LIN {X 0,Y 190.941,Z 458.891,A -85,B 0,C 180,E1 -21861.534,E2 -21861.534} C_VEL
LIN {X 0,Y 190.385,Z 460.614,A -85,B 0,C 180,E1 -21865.766,E2 -21865.766} C_VEL
LIN {X 0,Y 190.301,Z 461.211,A -85,B 0,C 180,E1 -21870,E2 -21870} C_VEL
LIN {X 0,Y 190.444,Z 460.499,A -85,B 0,C 180,E1 -21874.869,E2 -21874.869} C_VEL
LIN {X 0,Y 190.929,Z 458.975,A -85,B 0,C 180,E1 -21878.467,E2 -21878.467} C_VEL
LIN {X 0,Y 192.019,Z 456.147,A -85,B 0,C 180,E1 -21882.686,E2 -21882.686} C_VEL
LIN {X 0,Y 193.845,Z 452.093,A -85,B 0,C 180,E1 -21886.861,E2 -21886.861} C_VEL
LIN {X 0,Y 196.509,Z 446.712,A -85,B 0,C 180,E1 -21890.956,E2 -21890.956} C_VEL
LIN {X 0,Y 199.993,Z 439.849,A -85,B 0,C 180,E1 -21894.942,E2 -21894.942} C_VEL
LIN {X 0,Y 204.393,Z 431.274,A -85,B 0,C 180,E1 -21898.776,E2 -21898.776} C_VEL
LIN {X 0,Y 208.235,Z 423.562,A -85,B 0,C 180,E1 -21901.543,E2 -21901.543} C_VEL
LIN {X 0,Y 213.047,Z 412.865,A -85,B 0,C 180,E1 -21904.684,E2 -21904.684} C_VEL
LIN {X 0,Y 217.826,Z 401.819,A -85,B 0,C 180,E1 -21907.226,E2 -21907.226} C_VEL
LIN {X 0,Y 222.415,Z 389.72,A -85,B 0,C 180,E1 -21909.489,E2 -21909.489} C_VEL
LIN {X 0,Y 226.964,Z 376.424,A -85,B 0,C 180,E1 -21911.444,E2 -21911.444} C_VEL
LIN {X 0,Y 230.741,Z 362.87,A -85,B 0,C 180,E1 -21913.049,E2 -21913.049} C_VEL
LIN {X 0,Y 233.967,Z 349.116,A -85,B 0,C 180,E1 -21914.299,E2 -21914.299} C_VEL
LIN {X 0,Y 236.667,Z 334.427,A -85,B 0,C 180,E1 -21915.304,E2 -21915.304} C_VEL
LIN {X 0,Y 238.709,Z 319.352,A -85,B 0,C 180,E1 -21916.012,E2 -21916.012} C_VEL
LIN {X 0,Y 240.388,Z 297.392,A -85,B 0,C 180,E1 -21916.657,E2 -21916.657} C_VEL
LIN {X 0,Y 244.269,Z 236.804,A -85,B 0,C 180,E1 -21918.261,E2 -21918.261} C_VEL
LIN {X 0,Y 244.011,Z 235.536,A -85,B 0,C 180,E1 -21918.384,E2 -21918.384} C_VEL
LIN {X 0,Y 240.281,Z 227.752,A -85,B 0,C 180,E1 -21919.755,E2 -21919.755} C_VEL
LIN {X 0,Y 233.168,Z 215.506,A -85,B 0,C 180,E1 -21922.485,E2 -21922.485} C_VEL
LIN {X 0,Y 226.96,Z 205.762,A -85,B 0,C 180,E1 -21925.117,E2 -21925.117} C_VEL
LIN {X 0,Y 220.972,Z 197.115,A -85,B 0,C 180,E1 -21927.944,E2 -21927.944} C_VEL
LIN {X 0,Y 217.819,Z 192.871,A -85,B 0,C 180,E1 -21929.574,E2 -21929.574} C_VEL
LIN {X 0,Y 214.771,Z 188.838,A -85,B 0,C 180,E1 -21931.274,E2 -21931.274} C_VEL
LIN {X 0,Y 211.806,Z 184.879,A -85,B 0,C 180,E1 -21933.076,E2 -21933.076} C_VEL
LIN {X 0,Y 208.608,Z 181.315,A -85,B 0,C 180,E1 -21935.161,E2 -21935.161} C_VEL
LIN {X 0,Y 207.472,Z 179.38,A -85,B 0,C 180,E1 -21936.015,E2 -21936.015} C_VEL
LIN {X 0,Y 204.831,Z 177.101,A -85,B 0,C 180,E1 -21937.958,E2 -21937.958} C_VEL
LIN {X 0,Y 202.842,Z 173.863,A -85,B 0,C 180,E1 -21939.728,E2 -21939.728} C_VEL
LIN {X 0,Y 200.216,Z 171.989,A -85,B 0,C 180,E1 -21942.109,E2 -21942.109} C_VEL
LIN {X 0,Y 198.473,Z 169.066,A -85,B 0,C 180,E1 -21944.138,E2 -21944.138} C_VEL
LIN {X 0,Y 198.172,Z 168.139,A -85,B 0,C 180,E1 -21944.575,E2 -21944.575} C_VEL
LIN {X 0,Y 195.147,Z 166.479,A -85,B 0,C 180,E1 -21948.575,E2 -21948.575} C_VEL
LIN {X 0,Y 193.085,Z 162.801,A -85,B 0,C 180,E1 -21953.337,E2 -21953.337} C_VEL
LIN {X 0,Y 192.962,Z 162.066,A -85,B 0,C 180,E1 -21953.989,E2 -21953.989} C_VEL
LIN {X 0,Y 193.233,Z 162.041,A -85,B 0,C 180,E1 -21957.915,E2 -21957.915} C_VEL
LIN {X 0,Y 193.418,Z 162.001,A -85,B 0,C 180,E1 -21960,E2 -21960} C_VEL
LIN {X 0,Y 192.961,Z 162.06,A -85,B 0,C 180,E1 -21964.177,E2 -21964.177} C_VEL
LIN {X 0,Y 192.994,Z 162.232,A -85,B 0,C 180,E1 -21965.878,E2 -21965.878} C_VEL
LIN {X 0,Y 193.886,Z 164.688,A -85,B 0,C 180,E1 -21968.599,E2 -21968.599} C_VEL
LIN {X 0,Y 196.209,Z 167.297,A -85,B 0,C 180,E1 -21972.673,E2 -21972.673} C_VEL
LIN {X 0,Y 198.286,Z 168.3,A -85,B 0,C 180,E1 -21975.219,E2 -21975.219} C_VEL
LIN {X 0,Y 199.512,Z 170.977,A -85,B 0,C 180,E1 -21976.776,E2 -21976.776} C_VEL
LIN {X 0,Y 201.821,Z 173.285,A -85,B 0,C 180,E1 -21979.054,E2 -21979.054} C_VEL
LIN {X 0,Y 203.195,Z 174.283,A -85,B 0,C 180,E1 -21980.235,E2 -21980.235} C_VEL
LIN {X 0,Y 205.071,Z 177.346,A -85,B 0,C 180,E1 -21981.882,E2 -21981.882} C_VEL
LIN {X 0,Y 207.81,Z 179.895,A -85,B 0,C 180,E1 -21983.889,E2 -21983.889} C_VEL
LIN {X 0,Y 210.275,Z 183.372,A -85,B 0,C 180,E1 -21985.62,E2 -21985.62} C_VEL
LIN {X 0,Y 211.91,Z 185.069,A -85,B 0,C 180,E1 -21986.645,E2 -21986.645} C_VEL
LIN {X 0,Y 214.922,Z 189.001,A -85,B 0,C 180,E1 -21988.462,E2 -21988.462} C_VEL
LIN {X 0,Y 219.469,Z 195.238,A -85,B 0,C 180,E1 -21990.955,E2 -21990.955} C_VEL
LIN {X 0,Y 223.648,Z 202.088,A -85,B 0,C 180,E1 -21993.079,E2 -21993.079} C_VEL
LIN {X 0,Y 225.037,Z 204.616,A -85,B 0,C 180,E1 -21993.757,E2 -21993.757} C_VEL
LIN {X 0,Y 226.117,Z 207.654,A -85,B 0,C 180,E1 -21994.329,E2 -21994.329} C_VEL
LIN {X 0,Y 227.686,Z 214.53,A -85,B 0,C 180,E1 -21995.267,E2 -21995.267} C_VEL
LIN {X 0,Y 229.607,Z 223.383,A -85,B 0,C 180,E1 -21996.393,E2 -21996.393} C_VEL
LIN {X 0,Y 231.422,Z 228.024,A -85,B 0,C 180,E1 -21997.227,E2 -21997.227} C_VEL
LIN {X 0,Y 236.293,Z 238.89,A -85,B 0,C 180,E1 -21999.258,E2 -21999.258} C_VEL
LIN {X 0,Y 239.067,Z 245.621,A -85,B 0,C 180,E1 -22000.365,E2 -22000.365} C_VEL
LIN {X 0,Y 233.645,Z 325.426,A -85,B 0,C 180,E1 -22002.527,E2 -22002.527} C_VEL
LIN {X 0,Y 231.489,Z 341.56,A -85,B 0,C 180,E1 -22003.227,E2 -22003.227} C_VEL
LIN {X 0,Y 228.504,Z 356.805,A -85,B 0,C 180,E1 -22004.191,E2 -22004.191} C_VEL
LIN {X 0,Y 224.971,Z 370.535,A -85,B 0,C 180,E1 -22005.34,E2 -22005.34} C_VEL
LIN {X 0,Y 220.972,Z 384.002,A -85,B 0,C 180,E1 -22006.859,E2 -22006.859} C_VEL
LIN {X 0,Y 216.181,Z 397.756,A -85,B 0,C 180,E1 -22008.84,E2 -22008.84} C_VEL
LIN {X 0,Y 211.132,Z 410.12,A -85,B 0,C 180,E1 -22011.075,E2 -22011.075} C_VEL
LIN {X 0,Y 205.65,Z 422.297,A -85,B 0,C 180,E1 -22013.877,E2 -22013.877} C_VEL
LIN {X 0,Y 201.168,Z 431.703,A -85,B 0,C 180,E1 -22016.617,E2 -22016.617} C_VEL
LIN {X 0,Y 196.664,Z 440.962,A -85,B 0,C 180,E1 -22019.98,E2 -22019.98} C_VEL
LIN {X 0,Y 192.028,Z 449.677,A -85,B 0,C 180,E1 -22023.948,E2 -22023.948} C_VEL
LIN {X 0,Y 188.492,Z 456.683,A -85,B 0,C 180,E1 -22028.108,E2 -22028.108} C_VEL
LIN {X 0,Y 185.856,Z 462.197,A -85,B 0,C 180,E1 -22032.391,E2 -22032.391} C_VEL
LIN {X 0,Y 184.088,Z 466.373,A -85,B 0,C 180,E1 -22036.758,E2 -22036.758} C_VEL
LIN {X 0,Y 183.224,Z 469.308,A -85,B 0,C 180,E1 -22041.174,E2 -22041.174} C_VEL
LIN {X 0,Y 182.976,Z 471.063,A -85,B 0,C 180,E1 -22045.594,E2 -22045.594} C_VEL
LIN {X 0,Y 183.168,Z 471.669,A -85,B 0,C 180,E1 -22050,E2 -22050} C_VEL
LIN {X 0,Y 182.976,Z 471.047,A -85,B 0,C 180,E1 -22054.406,E2 -22054.406} C_VEL
LIN {X 0,Y 183.224,Z 469.271,A -85,B 0,C 180,E1 -22058.826,E2 -22058.826} C_VEL
LIN {X 0,Y 184.079,Z 466.319,A -85,B 0,C 180,E1 -22063.243,E2 -22063.243} C_VEL
LIN {X 0,Y 185.81,Z 462.128,A -85,B 0,C 180,E1 -22067.613,E2 -22067.613} C_VEL
LIN {X 0,Y 188.416,Z 456.587,A -85,B 0,C 180,E1 -22071.901,E2 -22071.901} C_VEL
LIN {X 0,Y 191.989,Z 449.551,A -85,B 0,C 180,E1 -22076.058,E2 -22076.058} C_VEL
LIN {X 0,Y 196.011,Z 442.038,A -85,B 0,C 180,E1 -22079.538,E2 -22079.538} C_VEL
LIN {X 0,Y 200.409,Z 432.978,A -85,B 0,C 180,E1 -22082.925,E2 -22082.925} C_VEL
LIN {X 0,Y 205.637,Z 422.094,A -85,B 0,C 180,E1 -22086.125,E2 -22086.125} C_VEL
LIN {X 0,Y 211.082,Z 409.864,A -85,B 0,C 180,E1 -22088.936,E2 -22088.936} C_VEL
LIN {X 0,Y 216.189,Z 397.432,A -85,B 0,C 180,E1 -22091.163,E2 -22091.163} C_VEL
LIN {X 0,Y 220.929,Z 383.607,A -85,B 0,C 180,E1 -22093.151,E2 -22093.151} C_VEL
LIN {X 0,Y 224.965,Z 370.042,A -85,B 0,C 180,E1 -22094.661,E2 -22094.661} C_VEL
LIN {X 0,Y 228.465,Z 356.243,A -85,B 0,C 180,E1 -22095.819,E2 -22095.819} C_VEL
LIN {X 0,Y 231.35,Z 341.579,A -85,B 0,C 180,E1 -22096.73,E2 -22096.73} C_VEL
LIN {X 0,Y 233.473,Z 325.428,A -85,B 0,C 180,E1 -22097.439,E2 -22097.439} C_VEL
LIN {X 0,Y 237.987,Z 259.996,A -85,B 0,C 180,E1 -22099.205,E2 -22099.205} C_VEL
LIN {X 0,Y 238.911,Z 245.472,A -85,B 0,C 180,E1 -22099.603,E2 -22099.603} C_VEL
LIN {X 0,Y 233.217,Z 231.952,A -85,B 0,C 180,E1 -22101.916,E2 -22101.916} C_VEL
LIN {X 0,Y 227.378,Z 220.017,A -85,B 0,C 180,E1 -22104.446,E2 -22104.446} C_VEL
LIN {X 0,Y 221.444,Z 208.914,A -85,B 0,C 180,E1 -22107.279,E2 -22107.279} C_VEL
LIN {X 0,Y 215.755,Z 199.426,A -85,B 0,C 180,E1 -22110.304,E2 -22110.304} C_VEL
LIN {X 0,Y 212.344,Z 194.903,A -85,B 0,C 180,E1 -22112.262,E2 -22112.262} C_VEL
LIN {X 0,Y 209.046,Z 190.532,A -85,B 0,C 180,E1 -22114.352,E2 -22114.352} C_VEL
LIN {X 0,Y 206.249,Z 187.049,A -85,B 0,C 180,E1 -22116.294,E2 -22116.294} C_VEL
LIN {X 0,Y 205.535,Z 185.913,A -85,B 0,C 180,E1 -22116.845,E2 -22116.845} C_VEL
LIN {X 0,Y 202.873,Z 183.255,A -85,B 0,C 180,E1 -22118.903,E2 -22118.903} C_VEL
LIN {X 0,Y 201.286,Z 180.606,A -85,B 0,C 180,E1 -22120.363,E2 -22120.363} C_VEL
LIN {X 0,Y 198.766,Z 178.632,A -85,B 0,C 180,E1 -22122.715,E2 -22122.715} C_VEL
LIN {X 0,Y 196.966,Z 175.504,A -85,B 0,C 180,E1 -22124.876,E2 -22124.876} C_VEL
LIN {X 0,Y 196.681,Z 175.002,A -85,B 0,C 180,E1 -22125.251,E2 -22125.251} C_VEL
LIN {X 0,Y 193.832,Z 173.17,A -85,B 0,C 180,E1 -22129.159,E2 -22129.159} C_VEL
LIN {X 0,Y 192.097,Z 169.801,A -85,B 0,C 180,E1 -22133.171,E2 -22133.171} C_VEL
LIN {X 0,Y 191.96,Z 169.223,A -85,B 0,C 180,E1 -22133.694,E2 -22133.694} C_VEL
LIN {X 0,Y 190.794,Z 168.603,A -85,B 0,C 180,E1 -22140,E2 -22140} C_VEL
LIN {X 0,Y 191.988,Z 169.275,A -85,B 0,C 180,E1 -22146.833,E2 -22146.833} C_VEL
LIN {X 0,Y 193.266,Z 172.44,A -85,B 0,C 180,E1 -22150.233,E2 -22150.233} C_VEL
LIN {X 0,Y 195.81,Z 174.67,A -85,B 0,C 180,E1 -22154.153,E2 -22154.153} C_VEL
LIN {X 0,Y 196.855,Z 175.279,A -85,B 0,C 180,E1 -22155.415,E2 -22155.415} C_VEL
LIN {X 0,Y 198.677,Z 178.613,A -85,B 0,C 180,E1 -22157.641,E2 -22157.641} C_VEL
LIN {X 0,Y 201.497,Z 180.984,A -85,B 0,C 180,E1 -22160.28,E2 -22160.28} C_VEL
LIN {X 0,Y 203.639,Z 184.293,A -85,B 0,C 180,E1 -22162.178,E2 -22162.178} C_VEL
LIN {X 0,Y 205.866,Z 186.424,A -85,B 0,C 180,E1 -22163.849,E2 -22163.849} C_VEL
LIN {X 0,Y 208.48,Z 190.012,A -85,B 0,C 180,E1 -22165.724,E2 -22165.724} C_VEL
LIN {X 0,Y 209.841,Z 191.608,A -85,B 0,C 180,E1 -22166.613,E2 -22166.613} C_VEL
LIN {X 0,Y 213.845,Z 196.934,A -85,B 0,C 180,E1 -22169.064,E2 -22169.064} C_VEL
LIN {X 0,Y 218.027,Z 202.706,A -85,B 0,C 180,E1 -22171.362,E2 -22171.362} C_VEL
LIN {X 0,Y 223.276,Z 210.46,A -85,B 0,C 180,E1 -22173.967,E2 -22173.967} C_VEL
LIN {X 0,Y 228.709,Z 219.049,A -85,B 0,C 180,E1 -22176.403,E2 -22176.403} C_VEL
LIN {X 0,Y 235.134,Z 230.2,A -85,B 0,C 180,E1 -22179.027,E2 -22179.027} C_VEL
LIN {X 0,Y 238.764,Z 237.398,A -85,B 0,C 180,E1 -22180.428,E2 -22180.428} C_VEL
LIN {X 0,Y 239.308,Z 238.724,A -85,B 0,C 180,E1 -22180.642,E2 -22180.642} C_VEL
LIN {X 0,Y 233.946,Z 317.1,A -85,B 0,C 180,E1 -22182.766,E2 -22182.766} C_VEL
LIN {X 0,Y 231.838,Z 333.001,A -85,B 0,C 180,E1 -22183.477,E2 -22183.477} C_VEL
LIN {X 0,Y 229.059,Z 348.105,A -85,B 0,C 180,E1 -22184.491,E2 -22184.491} C_VEL
LIN {X 0,Y 226.025,Z 361.087,A -85,B 0,C 180,E1 -22185.657,E2 -22185.657} C_VEL
LIN {X 0,Y 221.867,Z 375.842,A -85,B 0,C 180,E1 -22187.383,E2 -22187.383} C_VEL
LIN {X 0,Y 217.118,Z 389.289,A -85,B 0,C 180,E1 -22189.35,E2 -22189.35} C_VEL
LIN {X 0,Y 212.28,Z 401.491,A -85,B 0,C 180,E1 -22191.628,E2 -22191.628} C_VEL
LIN {X 0,Y 207.292,Z 412.609,A -85,B 0,C 180,E1 -22194.208,E2 -22194.208} C_VEL
LIN {X 0,Y 202.289,Z 423.39,A -85,B 0,C 180,E1 -22197.418,E2 -22197.418} C_VEL
LIN {X 0,Y 197.636,Z 432.347,A -85,B 0,C 180,E1 -22200.728,E2 -22200.728} C_VEL
LIN {X 0,Y 193.637,Z 439.764,A -85,B 0,C 180,E1 -22204.181,E2 -22204.181} C_VEL
LIN {X 0,Y 189.901,Z 446.69,A -85,B 0,C 180,E1 -22208.279,E2 -22208.279} C_VEL
LIN {X 0,Y 187.08,Z 452.124,A -85,B 0,C 180,E1 -22212.51,E2 -22212.51} C_VEL
LIN {X 0,Y 185.133,Z 456.219,A -85,B 0,C 180,E1 -22216.834,E2 -22216.834} C_VEL
LIN {X 0,Y 183.898,Z 459.091,A -85,B 0,C 180,E1 -22221.207,E2 -22221.207} C_VEL
LIN {X 0,Y 183.308,Z 460.812,A -85,B 0,C 180,E1 -22225.602,E2 -22225.602} C_VEL
LIN {X 0,Y 183.207,Z 461.41,A -85,B 0,C 180,E1 -22230,E2 -22230} C_VEL
LIN {X 0,Y 183.331,Z 460.795,A -85,B 0,C 180,E1 -22234.645,E2 -22234.645} C_VEL
LIN {X 0,Y 183.882,Z 459.174,A -85,B 0,C 180,E1 -22238.794,E2 -22238.794} C_VEL
LIN {X 0,Y 185.084,Z 456.345,A -85,B 0,C 180,E1 -22243.17,E2 -22243.17} C_VEL
LIN {X 0,Y 187.046,Z 452.292,A -85,B 0,C 180,E1 -22247.493,E2 -22247.493} C_VEL
LIN {X 0,Y 189.867,Z 446.91,A -85,B 0,C 180,E1 -22251.725,E2 -22251.725} C_VEL
LIN {X 0,Y 193.541,Z 440.048,A -85,B 0,C 180,E1 -22255.833,E2 -22255.833} C_VEL
LIN {X 0,Y 198.166,Z 431.472,A -85,B 0,C 180,E1 -22259.77,E2 -22259.77} C_VEL
LIN {X 0,Y 202.904,Z 422.349,A -85,B 0,C 180,E1 -22263.061,E2 -22263.061} C_VEL
LIN {X 0,Y 207.227,Z 413.062,A -85,B 0,C 180,E1 -22265.805,E2 -22265.805} C_VEL
LIN {X 0,Y 212.212,Z 402.015,A -85,B 0,C 180,E1 -22268.386,E2 -22268.386} C_VEL
LIN {X 0,Y 216.97,Z 389.915,A -85,B 0,C 180,E1 -22270.684,E2 -22270.684} C_VEL
LIN {X 0,Y 221.696,Z 376.618,A -85,B 0,C 180,E1 -22272.658,E2 -22272.658} C_VEL
LIN {X 0,Y 225.536,Z 363.341,A -85,B 0,C 180,E1 -22274.247,E2 -22274.247} C_VEL
LIN {X 0,Y 228.938,Z 349.308,A -85,B 0,C 180,E1 -22275.54,E2 -22275.54} C_VEL
LIN {X 0,Y 231.744,Z 334.615,A -85,B 0,C 180,E1 -22276.548,E2 -22276.548} C_VEL
LIN {X 0,Y 233.836,Z 319.536,A -85,B 0,C 180,E1 -22277.263,E2 -22277.263} C_VEL
LIN {X 0,Y 235.572,Z 297.567,A -85,B 0,C 180,E1 -22277.912,E2 -22277.912} C_VEL
LIN {X 0,Y 239.422,Z 238.711,A -85,B 0,C 180,E1 -22279.499,E2 -22279.499} C_VEL
LIN {X 0,Y 236.266,Z 232.138,A -85,B 0,C 180,E1 -22280.719,E2 -22280.719} C_VEL
LIN {X 0,Y 229.894,Z 220.899,A -85,B 0,C 180,E1 -22283.289,E2 -22283.289} C_VEL
LIN {X 0,Y 223.643,Z 210.885,A -85,B 0,C 180,E1 -22286.072,E2 -22286.072} C_VEL
LIN {X 0,Y 218.192,Z 202.869,A -85,B 0,C 180,E1 -22288.776,E2 -22288.776} C_VEL
LIN {X 0,Y 214.91,Z 198.382,A -85,B 0,C 180,E1 -22290.56,E2 -22290.56} C_VEL
LIN {X 0,Y 212.446,Z 194.999,A -85,B 0,C 180,E1 -22292.008,E2 -22292.008} C_VEL
LIN {X 0,Y 209.162,Z 190.651,A -85,B 0,C 180,E1 -22294.099,E2 -22294.099} C_VEL
LIN {X 0,Y 206.329,Z 187.196,A -85,B 0,C 180,E1 -22296.074,E2 -22296.074} C_VEL
LIN {X 0,Y 205.512,Z 185.922,A -85,B 0,C 180,E1 -22296.708,E2 -22296.708} C_VEL
LIN {X 0,Y 202.842,Z 183.268,A -85,B 0,C 180,E1 -22298.799,E2 -22298.799} C_VEL
LIN {X 0,Y 201.17,Z 180.617,A -85,B 0,C 180,E1 -22300.351,E2 -22300.351} C_VEL
LIN {X 0,Y 198.682,Z 178.546,A -85,B 0,C 180,E1 -22302.742,E2 -22302.742} C_VEL
LIN {X 0,Y 196.953,Z 175.539,A -85,B 0,C 180,E1 -22304.874,E2 -22304.874} C_VEL
LIN {X 0,Y 196.68,Z 175.004,A -85,B 0,C 180,E1 -22305.25,E2 -22305.25} C_VEL
LIN {X 0,Y 193.893,Z 173.218,A -85,B 0,C 180,E1 -22309.202,E2 -22309.202} C_VEL
LIN {X 0,Y 192.032,Z 169.492,A -85,B 0,C 180,E1 -22313.96,E2 -22313.96} C_VEL
LIN {X 0,Y 191.832,Z 169.072,A -85,B 0,C 180,E1 -22314.745,E2 -22314.745} C_VEL
LIN {X 0,Y 191.124,Z 168.711,A -85,B 0,C 180,E1 -22320,E2 -22320} C_VEL
LIN {X 0,Y 191.999,Z 169.276,A -85,B 0,C 180,E1 -22325.514,E2 -22325.514} C_VEL
LIN {X 0,Y 193.541,Z 172.705,A -85,B 0,C 180,E1 -22329.772,E2 -22329.772} C_VEL
LIN {X 0,Y 195.93,Z 174.681,A -85,B 0,C 180,E1 -22333.483,E2 -22333.483} C_VEL
LIN {X 0,Y 196.937,Z 175.325,A -85,B 0,C 180,E1 -22334.73,E2 -22334.73} C_VEL
LIN {X 0,Y 198.402,Z 178.102,A -85,B 0,C 180,E1 -22336.59,E2 -22336.59} C_VEL
LIN {X 0,Y 200.988,Z 180.461,A -85,B 0,C 180,E1 -22339.136,E2 -22339.136} C_VEL
LIN {X 0,Y 201.603,Z 181.112,A -85,B 0,C 180,E1 -22339.696,E2 -22339.696} C_VEL
LIN {X 0,Y 203.634,Z 184.207,A -85,B 0,C 180,E1 -22341.512,E2 -22341.512} C_VEL
LIN {X 0,Y 205.959,Z 186.478,A -85,B 0,C 180,E1 -22343.28,E2 -22343.28} C_VEL
LIN {X 0,Y 208.751,Z 190.265,A -85,B 0,C 180,E1 -22345.287,E2 -22345.287} C_VEL
LIN {X 0,Y 209.856,Z 191.516,A -85,B 0,C 180,E1 -22346.008,E2 -22346.008} C_VEL
LIN {X 0,Y 212.926,Z 195.511,A -85,B 0,C 180,E1 -22347.923,E2 -22347.923} C_VEL
LIN {X 0,Y 216.825,Z 201.138,A -85,B 0,C 180,E1 -22350.159,E2 -22350.159} C_VEL
LIN {X 0,Y 221.932,Z 209.649,A -85,B 0,C 180,E1 -22352.84,E2 -22352.84} C_VEL
LIN {X 0,Y 228.633,Z 222.323,A -85,B 0,C 180,E1 -22356.007,E2 -22356.007} C_VEL
LIN {X 0,Y 231.422,Z 228.024,A -85,B 0,C 180,E1 -22357.227,E2 -22357.227} C_VEL
LIN {X 0,Y 232.67,Z 231.012,A -85,B 0,C 180,E1 -22357.775,E2 -22357.775} C_VEL
LIN {X 0,Y 233.832,Z 236.24,A -85,B 0,C 180,E1 -22358.391,E2 -22358.391} C_VEL
LIN {X 0,Y 234.338,Z 243.95,A -85,B 0,C 180,E1 -22358.915,E2 -22358.915} C_VEL
LIN {X 0,Y 234.197,Z 250.053,A -85,B 0,C 180,E1 -22359.162,E2 -22359.162} C_VEL
LIN {X 0,Y 233.705,Z 258.247,A -85,B 0,C 180,E1 -22359.404,E2 -22359.404} C_VEL
LIN {X 0,Y 228.918,Z 325.244,A -85,B 0,C 180,E1 -22361.221,E2 -22361.221} C_VEL
LIN {X 0,Y 226.684,Z 341.371,A -85,B 0,C 180,E1 -22361.919,E2 -22361.919} C_VEL
LIN {X 0,Y 223.613,Z 356.613,A -85,B 0,C 180,E1 -22362.887,E2 -22362.887} C_VEL
LIN {X 0,Y 219.982,Z 370.343,A -85,B 0,C 180,E1 -22364.042,E2 -22364.042} C_VEL
LIN {X 0,Y 215.827,Z 383.807,A -85,B 0,C 180,E1 -22365.565,E2 -22365.565} C_VEL
LIN {X 0,Y 211.228,Z 396.609,A -85,B 0,C 180,E1 -22367.416,E2 -22367.416} C_VEL
LIN {X 0,Y 206.054,Z 408.85,A -85,B 0,C 180,E1 -22369.605,E2 -22369.605} C_VEL
LIN {X 0,Y 200.778,Z 420.337,A -85,B 0,C 180,E1 -22372.224,E2 -22372.224} C_VEL
LIN {X 0,Y 195.956,Z 430.01,A -85,B 0,C 180,E1 -22374.981,E2 -22374.981} C_VEL
LIN {X 0,Y 191.053,Z 439.537,A -85,B 0,C 180,E1 -22378.394,E2 -22378.394} C_VEL
LIN {X 0,Y 186.731,Z 447.447,A -85,B 0,C 180,E1 -22381.935,E2 -22381.935} C_VEL
LIN {X 0,Y 182.673,Z 454.855,A -85,B 0,C 180,E1 -22386.173,E2 -22386.173} C_VEL
LIN {X 0,Y 179.663,Z 460.741,A -85,B 0,C 180,E1 -22390.579,E2 -22390.579} C_VEL
LIN {X 0,Y 178.013,Z 464.247,A -85,B 0,C 180,E1 -22393.957,E2 -22393.957} C_VEL
LIN {X 0,Y 176.539,Z 467.791,A -85,B 0,C 180,E1 -22398.518,E2 -22398.518} C_VEL
LIN {X 0,Y 175.953,Z 470.131,A -85,B 0,C 180,E1 -22403.118,E2 -22403.118} C_VEL
LIN {X 0,Y 175.948,Z 471.312,A -85,B 0,C 180,E1 -22407.711,E2 -22407.711} C_VEL
LIN {X 0,Y 176.074,Z 471.47,A -85,B 0,C 180,E1 -22410,E2 -22410} C_VEL
LIN {X 0,Y 175.876,Z 470.848,A -85,B 0,C 180,E1 -22414.584,E2 -22414.584} C_VEL
LIN {X 0,Y 176.18,Z 469.071,A -85,B 0,C 180,E1 -22419.182,E2 -22419.182} C_VEL
LIN {X 0,Y 177.111,Z 466.117,A -85,B 0,C 180,E1 -22423.774,E2 -22423.774} C_VEL
LIN {X 0,Y 178.992,Z 461.926,A -85,B 0,C 180,E1 -22428.307,E2 -22428.307} C_VEL
LIN {X 0,Y 181.771,Z 456.385,A -85,B 0,C 180,E1 -22432.746,E2 -22432.746} C_VEL
LIN {X 0,Y 185.545,Z 449.348,A -85,B 0,C 180,E1 -22437.035,E2 -22437.035} C_VEL
LIN {X 0,Y 189.812,Z 441.835,A -85,B 0,C 180,E1 -22440.605,E2 -22440.605} C_VEL
LIN {X 0,Y 194.44,Z 432.772,A -85,B 0,C 180,E1 -22444.073,E2 -22444.073} C_VEL
LIN {X 0,Y 199.901,Z 421.891,A -85,B 0,C 180,E1 -22447.334,E2 -22447.334} C_VEL
LIN {X 0,Y 205.577,Z 409.661,A -85,B 0,C 180,E1 -22450.186,E2 -22450.186} C_VEL
LIN {X 0,Y 210.795,Z 397.457,A -85,B 0,C 180,E1 -22452.401,E2 -22452.401} C_VEL
LIN {X 0,Y 215.232,Z 385.084,A -85,B 0,C 180,E1 -22454.23,E2 -22454.23} C_VEL
LIN {X 0,Y 219.425,Z 371.68,A -85,B 0,C 180,E1 -22455.779,E2 -22455.779} C_VEL
LIN {X 0,Y 223.287,Z 357.175,A -85,B 0,C 180,E1 -22457.038,E2 -22457.038} C_VEL
LIN {X 0,Y 226.266,Z 342.898,A -85,B 0,C 180,E1 -22457.949,E2 -22457.949} C_VEL
LIN {X 0,Y 228.439,Z 327.549,A -85,B 0,C 180,E1 -22458.666,E2 -22458.666} C_VEL
LIN {X 0,Y 230.287,Z 305.152,A -85,B 0,C 180,E1 -22459.305,E2 -22459.305} C_VEL
LIN {X 0,Y 234.161,Z 247.952,A -85,B 0,C 180,E1 -22460.86,E2 -22460.86} C_VEL
LIN {X 0,Y 229.267,Z 236.183,A -85,B 0,C 180,E1 -22462.968,E2 -22462.968} C_VEL
LIN {X 0,Y 223.959,Z 224.989,A -85,B 0,C 180,E1 -22465.404,E2 -22465.404} C_VEL
LIN {X 0,Y 218.51,Z 214.435,A -85,B 0,C 180,E1 -22468.149,E2 -22468.149} C_VEL
LIN {X 0,Y 213.113,Z 205.24,A -85,B 0,C 180,E1 -22471.165,E2 -22471.165} C_VEL
LIN {X 0,Y 209.925,Z 200.885,A -85,B 0,C 180,E1 -22473.09,E2 -22473.09} C_VEL
LIN {X 0,Y 206.887,Z 196.776,A -85,B 0,C 180,E1 -22475.108,E2 -22475.108} C_VEL
LIN {X 0,Y 204.045,Z 192.972,A -85,B 0,C 180,E1 -22477.202,E2 -22477.202} C_VEL
LIN {X 0,Y 200.492,Z 188.777,A -85,B 0,C 180,E1 -22480.149,E2 -22480.149} C_VEL
LIN {X 0,Y 199.627,Z 187.312,A -85,B 0,C 180,E1 -22480.995,E2 -22480.995} C_VEL
LIN {X 0,Y 197.058,Z 184.978,A -85,B 0,C 180,E1 -22483.556,E2 -22483.556} C_VEL
LIN {X 0,Y 195.415,Z 181.895,A -85,B 0,C 180,E1 -22485.685,E2 -22485.685} C_VEL
LIN {X 0,Y 192.75,Z 180.074,A -85,B 0,C 180,E1 -22489.496,E2 -22489.496} C_VEL
LIN {X 0,Y 191.121,Z 176.83,A -85,B 0,C 180,E1 -22493.435,E2 -22493.435} C_VEL
LIN {X 0,Y 190.923,Z 176.143,A -85,B 0,C 180,E1 -22494.19,E2 -22494.19} C_VEL
LIN {X 0,Y 189.929,Z 175.647,A -85,B 0,C 180,E1 -22500,E2 -22500} C_VEL
LIN {X 0,Y 190.99,Z 176.244,A -85,B 0,C 180,E1 -22506.47,E2 -22506.47} C_VEL
LIN {X 0,Y 192.31,Z 179.543,A -85,B 0,C 180,E1 -22510.115,E2 -22510.115} C_VEL
LIN {X 0,Y 194.866,Z 181.71,A -85,B 0,C 180,E1 -22514.09,E2 -22514.09} C_VEL
LIN {X 0,Y 195.511,Z 182.204,A -85,B 0,C 180,E1 -22514.907,E2 -22514.907} C_VEL
LIN {X 0,Y 197.465,Z 185.548,A -85,B 0,C 180,E1 -22517.342,E2 -22517.342} C_VEL
LIN {X 0,Y 199.927,Z 187.783,A -85,B 0,C 180,E1 -22519.738,E2 -22519.738} C_VEL
LIN {X 0,Y 202.242,Z 191.188,A -85,B 0,C 180,E1 -22521.835,E2 -22521.835} C_VEL
LIN {X 0,Y 204.147,Z 193.178,A -85,B 0,C 180,E1 -22523.322,E2 -22523.322} C_VEL
LIN {X 0,Y 206.928,Z 196.849,A -85,B 0,C 180,E1 -22525.361,E2 -22525.361} C_VEL
LIN {X 0,Y 211.596,Z 203.222,A -85,B 0,C 180,E1 -22528.384,E2 -22528.384} C_VEL
LIN {X 0,Y 215.402,Z 208.544,A -85,B 0,C 180,E1 -22530.566,E2 -22530.566} C_VEL
LIN {X 0,Y 221.336,Z 217.573,A -85,B 0,C 180,E1 -22533.621,E2 -22533.621} C_VEL
LIN {X 0,Y 228.366,Z 229.35,A -85,B 0,C 180,E1 -22536.821,E2 -22536.821} C_VEL
LIN {X 0,Y 234.269,Z 240.502,A -85,B 0,C 180,E1 -22539.257,E2 -22539.257} C_VEL
LIN {X 0,Y 234.582,Z 241.219,A -85,B 0,C 180,E1 -22539.385,E2 -22539.385} C_VEL
LIN {X 0,Y 229.189,Z 317.356,A -85,B 0,C 180,E1 -22541.467,E2 -22541.467} C_VEL
LIN {X 0,Y 227.022,Z 333.21,A -85,B 0,C 180,E1 -22542.18,E2 -22542.18} C_VEL
LIN {X 0,Y 224.141,Z 348.311,A -85,B 0,C 180,E1 -22543.196,E2 -22543.196} C_VEL
LIN {X 0,Y 220.87,Z 361.856,A -85,B 0,C 180,E1 -22544.43,E2 -22544.43} C_VEL
LIN {X 0,Y 216.7,Z 376.045,A -85,B 0,C 180,E1 -22546.113,E2 -22546.113} C_VEL
LIN {X 0,Y 212.257,Z 388.25,A -85,B 0,C 180,E1 -22547.895,E2 -22547.895} C_VEL
LIN {X 0,Y 207.674,Z 399.591,A -85,B 0,C 180,E1 -22549.985,E2 -22549.985} C_VEL
LIN {X 0,Y 202.401,Z 411.044,A -85,B 0,C 180,E1 -22552.58,E2 -22552.58} C_VEL
LIN {X 0,Y 198.41,Z 419.318,A -85,B 0,C 180,E1 -22554.909,E2 -22554.909} C_VEL
LIN {X 0,Y 194.108,Z 427.628,A -85,B 0,C 180,E1 -22557.721,E2 -22557.721} C_VEL
LIN {X 0,Y 189.557,Z 435.88,A -85,B 0,C 180,E1 -22561.185,E2 -22561.185} C_VEL
LIN {X 0,Y 185.117,Z 443.627,A -85,B 0,C 180,E1 -22565.316,E2 -22565.316} C_VEL
LIN {X 0,Y 181.758,Z 449.781,A -85,B 0,C 180,E1 -22569.635,E2 -22569.635} C_VEL
LIN {X 0,Y 179.098,Z 454.532,A -85,B 0,C 180,E1 -22574.057,E2 -22574.057} C_VEL
LIN {X 0,Y 177.457,Z 458.002,A -85,B 0,C 180,E1 -22578.579,E2 -22578.579} C_VEL
LIN {X 0,Y 176.468,Z 460.292,A -85,B 0,C 180,E1 -22583.138,E2 -22583.138} C_VEL
LIN {X 0,Y 176.106,Z 461.454,A -85,B 0,C 180,E1 -22587.713,E2 -22587.713} C_VEL
LIN {X 0,Y 176.116,Z 461.608,A -85,B 0,C 180,E1 -22590,E2 -22590} C_VEL
LIN {X 0,Y 176.226,Z 461.047,A -85,B 0,C 180,E1 -22594.575,E2 -22594.575} C_VEL
LIN {X 0,Y 176.85,Z 459.373,A -85,B 0,C 180,E1 -22599.147,E2 -22599.147} C_VEL
LIN {X 0,Y 178.133,Z 456.545,A -85,B 0,C 180,E1 -22603.693,E2 -22603.693} C_VEL
LIN {X 0,Y 180.274,Z 452.49,A -85,B 0,C 180,E1 -22608.173,E2 -22608.173} C_VEL
LIN {X 0,Y 183.248,Z 447.109,A -85,B 0,C 180,E1 -22612.552,E2 -22612.552} C_VEL
LIN {X 0,Y 187.161,Z 440.245,A -85,B 0,C 180,E1 -22616.783,E2 -22616.783} C_VEL
LIN {X 0,Y 191.992,Z 431.67,A -85,B 0,C 180,E1 -22620.829,E2 -22620.829} C_VEL
LIN {X 0,Y 196.967,Z 422.547,A -85,B 0,C 180,E1 -22624.193,E2 -22624.193} C_VEL
LIN {X 0,Y 201.489,Z 413.259,A -85,B 0,C 180,E1 -22626.991,E2 -22626.991} C_VEL
LIN {X 0,Y 206.674,Z 402.211,A -85,B 0,C 180,E1 -22629.613,E2 -22629.613} C_VEL
LIN {X 0,Y 211.634,Z 390.11,A -85,B 0,C 180,E1 -22631.938,E2 -22631.938} C_VEL
LIN {X 0,Y 216.536,Z 376.812,A -85,B 0,C 180,E1 -22633.929,E2 -22633.929} C_VEL
LIN {X 0,Y 220.442,Z 363.775,A -85,B 0,C 180,E1 -22635.507,E2 -22635.507} C_VEL
LIN {X 0,Y 224.036,Z 349.499,A -85,B 0,C 180,E1 -22636.833,E2 -22636.833} C_VEL
LIN {X 0,Y 226.918,Z 334.804,A -85,B 0,C 180,E1 -22637.85,E2 -22637.85} C_VEL
LIN {X 0,Y 229.094,Z 319.719,A -85,B 0,C 180,E1 -22638.563,E2 -22638.563} C_VEL
LIN {X 0,Y 230.879,Z 297.742,A -85,B 0,C 180,E1 -22639.218,E2 -22639.218} C_VEL
LIN {X 0,Y 234.734,Z 241.966,A -85,B 0,C 180,E1 -22640.712,E2 -22640.712} C_VEL
LIN {X 0,Y 234.352,Z 240.49,A -85,B 0,C 180,E1 -22640.897,E2 -22640.897} C_VEL
LIN {X 0,Y 228.438,Z 229.366,A -85,B 0,C 180,E1 -22643.344,E2 -22643.344} C_VEL
LIN {X 0,Y 222.221,Z 218.909,A -85,B 0,C 180,E1 -22646.164,E2 -22646.164} C_VEL
LIN {X 0,Y 216.074,Z 209.372,A -85,B 0,C 180,E1 -22649.302,E2 -22649.302} C_VEL
LIN {X 0,Y 210.515,Z 201.549,A -85,B 0,C 180,E1 -22652.54,E2 -22652.54} C_VEL
LIN {X 0,Y 206.871,Z 196.781,A -85,B 0,C 180,E1 -22654.949,E2 -22654.949} C_VEL
LIN {X 0,Y 204.106,Z 193.061,A -85,B 0,C 180,E1 -22657.008,E2 -22657.008} C_VEL
LIN {X 0,Y 200.775,Z 189.193,A -85,B 0,C 180,E1 -22659.777,E2 -22659.777} C_VEL
LIN {X 0,Y 199.797,Z 187.472,A -85,B 0,C 180,E1 -22660.745,E2 -22660.745} C_VEL
LIN {X 0,Y 197.24,Z 185.21,A -85,B 0,C 180,E1 -22663.305,E2 -22663.305} C_VEL
LIN {X 0,Y 195.422,Z 181.921,A -85,B 0,C 180,E1 -22665.685,E2 -22665.685} C_VEL
LIN {X 0,Y 192.728,Z 180,A -85,B 0,C 180,E1 -22669.719,E2 -22669.719} C_VEL
LIN {X 0,Y 190.969,Z 176.133,A -85,B 0,C 180,E1 -22674.721,E2 -22674.721} C_VEL
LIN {X 0,Y 190.261,Z 175.735,A -85,B 0,C 180,E1 -22680,E2 -22680} C_VEL
LIN {X 0,Y 191.022,Z 176.229,A -85,B 0,C 180,E1 -22685.145,E2 -22685.145} C_VEL
LIN {X 0,Y 192.773,Z 180.034,A -85,B 0,C 180,E1 -22690.015,E2 -22690.015} C_VEL
LIN {X 0,Y 195.57,Z 182.152,A -85,B 0,C 180,E1 -22694.171,E2 -22694.171} C_VEL
LIN {X 0,Y 197.313,Z 185.245,A -85,B 0,C 180,E1 -22696.422,E2 -22696.422} C_VEL
LIN {X 0,Y 199.93,Z 187.705,A -85,B 0,C 180,E1 -22699.042,E2 -22699.042} C_VEL
LIN {X 0,Y 202.344,Z 191.249,A -85,B 0,C 180,E1 -22701.255,E2 -22701.255} C_VEL
LIN {X 0,Y 204.183,Z 193.148,A -85,B 0,C 180,E1 -22702.702,E2 -22702.702} C_VEL
LIN {X 0,Y 207.111,Z 197.008,A -85,B 0,C 180,E1 -22704.863,E2 -22704.863} C_VEL
LIN {X 0,Y 211.677,Z 203.215,A -85,B 0,C 180,E1 -22707.833,E2 -22707.833} C_VEL
LIN {X 0,Y 214.246,Z 207.035,A -85,B 0,C 180,E1 -22709.354,E2 -22709.354} C_VEL
LIN {X 0,Y 219.182,Z 215.62,A -85,B 0,C 180,E1 -22712.078,E2 -22712.078} C_VEL
LIN {X 0,Y 225.298,Z 227.459,A -85,B 0,C 180,E1 -22715.11,E2 -22715.11} C_VEL
LIN {X 0,Y 230.971,Z 239.836,A -85,B 0,C 180,E1 -22717.671,E2 -22717.671} C_VEL
LIN {X 0,Y 234.337,Z 248.108,A -85,B 0,C 180,E1 -22719.112,E2 -22719.112} C_VEL
LIN {X 0,Y 233.705,Z 258.247,A -85,B 0,C 180,E1 -22719.404,E2 -22719.404} C_VEL
LIN {X 0,Y 232.889,Z 264.099,A -85,B 0,C 180,E1 -22719.438,E2 -22719.438} C_VEL
LIN {X 0,Y 227.867,Z 283.155,A -85,B 0,C 180,E1 -22718.831,E2 -22718.831} C_VEL
LIN {X 0,Y 227.049,Z 289.008,A -85,B 0,C 180,E1 -22718.865,E2 -22718.865} C_VEL
LIN {X 0,Y 224.148,Z 326.247,A -85,B 0,C 180,E1 -22719.896,E2 -22719.896} C_VEL
LIN {X 0,Y 221.853,Z 341.944,A -85,B 0,C 180,E1 -22720.597,E2 -22720.597} C_VEL
LIN {X 0,Y 218.838,Z 356.421,A -85,B 0,C 180,E1 -22721.523,E2 -22721.523} C_VEL
LIN {X 0,Y 215.106,Z 370.15,A -85,B 0,C 180,E1 -22722.682,E2 -22722.682} C_VEL
LIN {X 0,Y 210.802,Z 383.606,A -85,B 0,C 180,E1 -22724.209,E2 -22724.209} C_VEL
LIN {X 0,Y 205.903,Z 396.751,A -85,B 0,C 180,E1 -22726.128,E2 -22726.128} C_VEL
LIN {X 0,Y 200.192,Z 409.726,A -85,B 0,C 180,E1 -22728.499,E2 -22728.499} C_VEL
LIN {X 0,Y 194.295,Z 421.902,A -85,B 0,C 180,E1 -22731.393,E2 -22731.393} C_VEL
LIN {X 0,Y 189.353,Z 431.305,A -85,B 0,C 180,E1 -22734.227,E2 -22734.227} C_VEL
LIN {X 0,Y 184.331,Z 440.563,A -85,B 0,C 180,E1 -22737.739,E2 -22737.739} C_VEL
LIN {X 0,Y 179.825,Z 448.263,A -85,B 0,C 180,E1 -22741.395,E2 -22741.395} C_VEL
LIN {X 0,Y 176.128,Z 454.655,A -85,B 0,C 180,E1 -22745.23,E2 -22745.23} C_VEL
LIN {X 0,Y 172.91,Z 460.541,A -85,B 0,C 180,E1 -22749.788,E2 -22749.788} C_VEL
LIN {X 0,Y 171.142,Z 464.047,A -85,B 0,C 180,E1 -22753.294,E2 -22753.294} C_VEL
LIN {X 0,Y 169.541,Z 467.592,A -85,B 0,C 180,E1 -22758.038,E2 -22758.038} C_VEL
LIN {X 0,Y 168.884,Z 469.932,A -85,B 0,C 180,E1 -22762.828,E2 -22762.828} C_VEL
LIN {X 0,Y 168.857,Z 471.114,A -85,B 0,C 180,E1 -22767.614,E2 -22767.614} C_VEL
LIN {X 0,Y 168.983,Z 471.272,A -85,B 0,C 180,E1 -22770,E2 -22770} C_VEL
LIN {X 0,Y 168.792,Z 470.649,A -85,B 0,C 180,E1 -22774.777,E2 -22774.777} C_VEL
LIN {X 0,Y 169.122,Z 468.87,A -85,B 0,C 180,E1 -22779.568,E2 -22779.568} C_VEL
LIN {X 0,Y 170.159,Z 465.916,A -85,B 0,C 180,E1 -22784.348,E2 -22784.348} C_VEL
LIN {X 0,Y 172.2,Z 461.724,A -85,B 0,C 180,E1 -22789.057,E2 -22789.057} C_VEL
LIN {X 0,Y 175.193,Z 456.183,A -85,B 0,C 180,E1 -22793.651,E2 -22793.651} C_VEL
LIN {X 0,Y 179.17,Z 449.145,A -85,B 0,C 180,E1 -22798.08,E2 -22798.08} C_VEL
LIN {X 0,Y 183.659,Z 441.632,A -85,B 0,C 180,E1 -22801.747,E2 -22801.747} C_VEL
LIN {X 0,Y 188.557,Z 432.57,A -85,B 0,C 180,E1 -22805.291,E2 -22805.291} C_VEL
LIN {X 0,Y 194.266,Z 421.688,A -85,B 0,C 180,E1 -22808.613,E2 -22808.613} C_VEL
LIN {X 0,Y 200.183,Z 409.458,A -85,B 0,C 180,E1 -22811.503,E2 -22811.503} C_VEL
LIN {X 0,Y 205.507,Z 397.475,A -85,B 0,C 180,E1 -22813.703,E2 -22813.703} C_VEL
LIN {X 0,Y 210.243,Z 384.733,A -85,B 0,C 180,E1 -22815.604,E2 -22815.604} C_VEL
LIN {X 0,Y 214.533,Z 371.475,A -85,B 0,C 180,E1 -22817.138,E2 -22817.138} C_VEL
LIN {X 0,Y 218.214,Z 358.099,A -85,B 0,C 180,E1 -22818.314,E2 -22818.314} C_VEL
LIN {X 0,Y 221.414,Z 343.452,A -85,B 0,C 180,E1 -22819.273,E2 -22819.273} C_VEL
LIN {X 0,Y 223.658,Z 328.605,A -85,B 0,C 180,E1 -22819.981,E2 -22819.981} C_VEL
LIN {X 0,Y 225.306,Z 310.699,A -85,B 0,C 180,E1 -22820.517,E2 -22820.517} C_VEL
LIN {X 0,Y 229.552,Z 250.424,A -85,B 0,C 180,E1 -22822.161,E2 -22822.161} C_VEL
LIN {X 0,Y 224.316,Z 237.822,A -85,B 0,C 180,E1 -22824.576,E2 -22824.576} C_VEL
LIN {X 0,Y 218.812,Z 226.263,A -85,B 0,C 180,E1 -22827.317,E2 -22827.317} C_VEL
LIN {X 0,Y 214.601,Z 218.218,A -85,B 0,C 180,E1 -22829.611,E2 -22829.611} C_VEL
LIN {X 0,Y 210.489,Z 211.039,A -85,B 0,C 180,E1 -22832.064,E2 -22832.064} C_VEL
LIN {X 0,Y 207.616,Z 206.971,A -85,B 0,C 180,E1 -22833.892,E2 -22833.892} C_VEL
LIN {X 0,Y 204.78,Z 203.057,A -85,B 0,C 180,E1 -22835.869,E2 -22835.869} C_VEL
LIN {X 0,Y 201.585,Z 198.754,A -85,B 0,C 180,E1 -22838.36,E2 -22838.36} C_VEL
LIN {X 0,Y 198.72,Z 195.126,A -85,B 0,C 180,E1 -22840.905,E2 -22840.905} C_VEL
LIN {X 0,Y 197.997,Z 193.989,A -85,B 0,C 180,E1 -22841.638,E2 -22841.638} C_VEL
LIN {X 0,Y 195.457,Z 191.386,A -85,B 0,C 180,E1 -22844.337,E2 -22844.337} C_VEL
LIN {X 0,Y 194.153,Z 188.837,A -85,B 0,C 180,E1 -22846.125,E2 -22846.125} C_VEL
LIN {X 0,Y 191.471,Z 186.734,A -85,B 0,C 180,E1 -22850.226,E2 -22850.226} C_VEL
LIN {X 0,Y 189.999,Z 183.333,A -85,B 0,C 180,E1 -22854.295,E2 -22854.295} C_VEL
LIN {X 0,Y 189.064,Z 182.695,A -85,B 0,C 180,E1 -22860,E2 -22860} C_VEL
LIN {X 0,Y 190.029,Z 183.348,A -85,B 0,C 180,E1 -22866.237,E2 -22866.237} C_VEL
LIN {X 0,Y 191.382,Z 186.672,A -85,B 0,C 180,E1 -22870.046,E2 -22870.046} C_VEL
LIN {X 0,Y 194.201,Z 189.083,A -85,B 0,C 180,E1 -22874.407,E2 -22874.407} C_VEL
LIN {X 0,Y 196.153,Z 192.368,A -85,B 0,C 180,E1 -22876.925,E2 -22876.925} C_VEL
LIN {X 0,Y 198.33,Z 194.443,A -85,B 0,C 180,E1 -22879.134,E2 -22879.134} C_VEL
LIN {X 0,Y 200.924,Z 198.166,A -85,B 0,C 180,E1 -22881.548,E2 -22881.548} C_VEL
LIN {X 0,Y 202.307,Z 199.678,A -85,B 0,C 180,E1 -22882.668,E2 -22882.668} C_VEL
LIN {X 0,Y 206.042,Z 204.839,A -85,B 0,C 180,E1 -22885.477,E2 -22885.477} C_VEL
LIN {X 0,Y 209.557,Z 209.722,A -85,B 0,C 180,E1 -22887.8,E2 -22887.8} C_VEL
LIN {X 0,Y 213.966,Z 216.094,A -85,B 0,C 180,E1 -22890.401,E2 -22890.401} C_VEL
LIN {X 0,Y 220.324,Z 226.292,A -85,B 0,C 180,E1 -22893.727,E2 -22893.727} C_VEL
LIN {X 0,Y 226.622,Z 237.541,A -85,B 0,C 180,E1 -22896.653,E2 -22896.653} C_VEL
LIN {X 0,Y 229.941,Z 243.971,A -85,B 0,C 180,E1 -22898.081,E2 -22898.081} C_VEL
LIN {X 0,Y 224.607,Z 317.241,A -85,B 0,C 180,E1 -22900.103,E2 -22900.103} C_VEL
LIN {X 0,Y 222.447,Z 332.646,A -85,B 0,C 180,E1 -22900.776,E2 -22900.776} C_VEL
LIN {X 0,Y 219.611,Z 347.36,A -85,B 0,C 180,E1 -22901.751,E2 -22901.751} C_VEL
LIN {X 0,Y 216.04,Z 361.776,A -85,B 0,C 180,E1 -22903.056,E2 -22903.056} C_VEL
LIN {X 0,Y 211.648,Z 376.249,A -85,B 0,C 180,E1 -22904.783,E2 -22904.783} C_VEL
LIN {X 0,Y 206.556,Z 389.694,A -85,B 0,C 180,E1 -22906.784,E2 -22906.784} C_VEL
LIN {X 0,Y 201.324,Z 401.896,A -85,B 0,C 180,E1 -22909.115,E2 -22909.115} C_VEL
LIN {X 0,Y 195.936,Z 413.012,A -85,B 0,C 180,E1 -22911.776,E2 -22911.776} C_VEL
LIN {X 0,Y 191.914,Z 420.875,A -85,B 0,C 180,E1 -22914.131,E2 -22914.131} C_VEL
LIN {X 0,Y 187.39,Z 429.092,A -85,B 0,C 180,E1 -22917.056,E2 -22917.056} C_VEL
LIN {X 0,Y 182.733,Z 437.166,A -85,B 0,C 180,E1 -22920.635,E2 -22920.635} C_VEL
LIN {X 0,Y 178.647,Z 443.828,A -85,B 0,C 180,E1 -22924.358,E2 -22924.358} C_VEL
LIN {X 0,Y 175.084,Z 449.982,A -85,B 0,C 180,E1 -22928.822,E2 -22928.822} C_VEL
LIN {X 0,Y 172.241,Z 454.733,A -85,B 0,C 180,E1 -22933.404,E2 -22933.404} C_VEL
LIN {X 0,Y 170.492,Z 458.202,A -85,B 0,C 180,E1 -22938.106,E2 -22938.106} C_VEL
LIN {X 0,Y 169.422,Z 460.491,A -85,B 0,C 180,E1 -22942.851,E2 -22942.851} C_VEL
LIN {X 0,Y 169.01,Z 461.653,A -85,B 0,C 180,E1 -22947.617,E2 -22947.617} C_VEL
LIN {X 0,Y 169.027,Z 461.807,A -85,B 0,C 180,E1 -22950,E2 -22950} C_VEL
LIN {X 0,Y 169.147,Z 461.245,A -85,B 0,C 180,E1 -22954.767,E2 -22954.767} C_VEL
LIN {X 0,Y 169.841,Z 459.571,A -85,B 0,C 180,E1 -22959.528,E2 -22959.528} C_VEL
LIN {X 0,Y 171.199,Z 456.744,A -85,B 0,C 180,E1 -22964.259,E2 -22964.259} C_VEL
LIN {X 0,Y 173.529,Z 452.688,A -85,B 0,C 180,E1 -22968.905,E2 -22968.905} C_VEL
LIN {X 0,Y 176.675,Z 447.308,A -85,B 0,C 180,E1 -22973.441,E2 -22973.441} C_VEL
LIN {X 0,Y 180.808,Z 440.444,A -85,B 0,C 180,E1 -22977.804,E2 -22977.804} C_VEL
LIN {X 0,Y 185.893,Z 431.868,A -85,B 0,C 180,E1 -22981.958,E2 -22981.958} C_VEL
LIN {X 0,Y 191.097,Z 422.744,A -85,B 0,C 180,E1 -22985.397,E2 -22985.397} C_VEL
LIN {X 0,Y 195.839,Z 413.456,A -85,B 0,C 180,E1 -22988.247,E2 -22988.247} C_VEL
LIN {X 0,Y 201.705,Z 401.415,A -85,B 0,C 180,E1 -22991.122,E2 -22991.122} C_VEL
LIN {X 0,Y 206.926,Z 389.118,A -85,B 0,C 180,E1 -22993.454,E2 -22993.454} C_VEL
LIN {X 0,Y 211.974,Z 375.591,A -85,B 0,C 180,E1 -22995.455,E2 -22995.455} C_VEL
LIN {X 0,Y 216.041,Z 362.198,A -85,B 0,C 180,E1 -22997.049,E2 -22997.049} C_VEL
LIN {X 0,Y 219.795,Z 347.408,A -85,B 0,C 180,E1 -22998.368,E2 -22998.368} C_VEL
LIN {X 0,Y 222.786,Z 331.84,A -85,B 0,C 180,E1 -22999.383,E2 -22999.383} C_VEL
LIN {X 0,Y 224.904,Z 316.297,A -85,B 0,C 180,E1 -23000.048,E2 -23000.048} C_VEL
LIN {X 0,Y 230.128,Z 244.116,A -85,B 0,C 180,E1 -23002.037,E2 -23002.037} C_VEL
LIN {X 0,Y 223.723,Z 232.084,A -85,B 0,C 180,E1 -23004.861,E2 -23004.861} C_VEL
LIN {X 0,Y 217.994,Z 222.411,A -85,B 0,C 180,E1 -23007.658,E2 -23007.658} C_VEL
LIN {X 0,Y 212.873,Z 214.475,A -85,B 0,C 180,E1 -23010.451,E2 -23010.451} C_VEL
LIN {X 0,Y 209.884,Z 210.134,A -85,B 0,C 180,E1 -23012.247,E2 -23012.247} C_VEL
LIN {X 0,Y 207.551,Z 206.865,A -85,B 0,C 180,E1 -23013.758,E2 -23013.758} C_VEL
LIN {X 0,Y 204.965,Z 203.251,A -85,B 0,C 180,E1 -23015.578,E2 -23015.578} C_VEL
LIN {X 0,Y 201.626,Z 198.805,A -85,B 0,C 180,E1 -23018.195,E2 -23018.195} C_VEL
LIN {X 0,Y 199.005,Z 195.556,A -85,B 0,C 180,E1 -23020.531,E2 -23020.531} C_VEL
LIN {X 0,Y 197.916,Z 193.987,A -85,B 0,C 180,E1 -23021.63,E2 -23021.63} C_VEL
LIN {X 0,Y 195.426,Z 191.352,A -85,B 0,C 180,E1 -23024.352,E2 -23024.352} C_VEL
LIN {X 0,Y 193.981,Z 188.747,A -85,B 0,C 180,E1 -23026.379,E2 -23026.379} C_VEL
LIN {X 0,Y 191.458,Z 186.626,A -85,B 0,C 180,E1 -23030.492,E2 -23030.492} C_VEL
LIN {X 0,Y 189.963,Z 183.139,A -85,B 0,C 180,E1 -23035.225,E2 -23035.225} C_VEL
LIN {X 0,Y 189.399,Z 182.762,A -85,B 0,C 180,E1 -23040,E2 -23040} C_VEL
LIN {X 0,Y 190.068,Z 183.306,A -85,B 0,C 180,E1 -23044.872,E2 -23044.872} C_VEL
LIN {X 0,Y 191.804,Z 187.069,A -85,B 0,C 180,E1 -23049.861,E2 -23049.861} C_VEL
LIN {X 0,Y 194.268,Z 189.044,A -85,B 0,C 180,E1 -23053.667,E2 -23053.667} C_VEL
LIN {X 0,Y 196.335,Z 192.484,A -85,B 0,C 180,E1 -23056.373,E2 -23056.373} C_VEL
LIN {X 0,Y 198.377,Z 194.439,A -85,B 0,C 180,E1 -23058.472,E2 -23058.472} C_VEL
LIN {X 0,Y 201.067,Z 198.221,A -85,B 0,C 180,E1 -23060.994,E2 -23060.994} C_VEL
LIN {X 0,Y 202.365,Z 199.66,A -85,B 0,C 180,E1 -23062.056,E2 -23062.056} C_VEL
LIN {X 0,Y 206.221,Z 205.002,A -85,B 0,C 180,E1 -23064.978,E2 -23064.978} C_VEL
LIN {X 0,Y 209.64,Z 209.726,A -85,B 0,C 180,E1 -23067.246,E2 -23067.246} C_VEL
LIN {X 0,Y 211.785,Z 213.065,A -85,B 0,C 180,E1 -23068.576,E2 -23068.576} C_VEL
LIN {X 0,Y 216.574,Z 221.699,A -85,B 0,C 180,E1 -23071.347,E2 -23071.347} C_VEL
LIN {X 0,Y 222.011,Z 232.682,A -85,B 0,C 180,E1 -23074.187,E2 -23074.187} C_VEL
LIN {X 0,Y 227.265,Z 244.409,A -85,B 0,C 180,E1 -23076.688,E2 -23076.688} C_VEL
LIN {X 0,Y 229.72,Z 250.598,A -85,B 0,C 180,E1 -23077.806,E2 -23077.806} C_VEL
LIN {X 0,Y 227.049,Z 289.008,A -85,B 0,C 180,E1 -23078.865,E2 -23078.865} C_VEL
LIN {X 0,Y 226.231,Z 294.865,A -85,B 0,C 180,E1 -23078.892,E2 -23078.892} C_VEL
LIN {X 0,Y 221.185,Z 313.91,A -85,B 0,C 180,E1 -23078.228,E2 -23078.228} C_VEL
LIN {X 0,Y 220.316,Z 319.749,A -85,B 0,C 180,E1 -23078.283,E2 -23078.283} C_VEL
LIN {X 0,Y 218.463,Z 334.874,A -85,B 0,C 180,E1 -23078.837,E2 -23078.837} C_VEL
LIN {X 0,Y 215.653,Z 349.829,A -85,B 0,C 180,E1 -23079.653,E2 -23079.653} C_VEL
LIN {X 0,Y 212.091,Z 363.991,A -85,B 0,C 180,E1 -23080.711,E2 -23080.711} C_VEL
LIN {X 0,Y 208.084,Z 377.05,A -85,B 0,C 180,E1 -23082.008,E2 -23082.008} C_VEL
LIN {X 0,Y 203.213,Z 390.542,A -85,B 0,C 180,E1 -23083.764,E2 -23083.764} C_VEL
LIN {X 0,Y 197.977,Z 403.03,A -85,B 0,C 180,E1 -23085.839,E2 -23085.839} C_VEL
LIN {X 0,Y 192.488,Z 414.459,A -85,B 0,C 180,E1 -23088.215,E2 -23088.215} C_VEL
LIN {X 0,Y 186.975,Z 424.975,A -85,B 0,C 180,E1 -23090.979,E2 -23090.979} C_VEL
LIN {X 0,Y 181.989,Z 433.904,A -85,B 0,C 180,E1 -23093.919,E2 -23093.919} C_VEL
LIN {X 0,Y 176.952,Z 442.707,A -85,B 0,C 180,E1 -23097.576,E2 -23097.576} C_VEL
LIN {X 0,Y 172.928,Z 449.079,A -85,B 0,C 180,E1 -23100.811,E2 -23100.811} C_VEL
LIN {X 0,Y 168.684,Z 456.083,A -85,B 0,C 180,E1 -23105.377,E2 -23105.377} C_VEL
LIN {X 0,Y 165.501,Z 461.598,A -85,B 0,C 180,E1 -23110.14,E2 -23110.14} C_VEL
LIN {X 0,Y 163.249,Z 465.773,A -85,B 0,C 180,E1 -23115.03,E2 -23115.03} C_VEL
LIN {X 0,Y 162.086,Z 468.71,A -85,B 0,C 180,E1 -23120.012,E2 -23120.012} C_VEL
LIN {X 0,Y 161.705,Z 470.466,A -85,B 0,C 180,E1 -23125.013,E2 -23125.013} C_VEL
LIN {X 0,Y 161.894,Z 471.073,A -85,B 0,C 180,E1 -23130,E2 -23130} C_VEL
LIN {X 0,Y 161.705,Z 470.449,A -85,B 0,C 180,E1 -23134.987,E2 -23134.987} C_VEL
LIN {X 0,Y 162.085,Z 468.67,A -85,B 0,C 180,E1 -23139.988,E2 -23139.988} C_VEL
LIN {X 0,Y 163.233,Z 465.715,A -85,B 0,C 180,E1 -23144.971,E2 -23144.971} C_VEL
LIN {X 0,Y 165.442,Z 461.523,A -85,B 0,C 180,E1 -23149.867,E2 -23149.867} C_VEL
LIN {X 0,Y 168.639,Z 455.981,A -85,B 0,C 180,E1 -23154.629,E2 -23154.629} C_VEL
LIN {X 0,Y 172.876,Z 448.942,A -85,B 0,C 180,E1 -23159.199,E2 -23159.199} C_VEL
LIN {X 0,Y 177.57,Z 441.429,A -85,B 0,C 180,E1 -23162.971,E2 -23162.971} C_VEL
LIN {X 0,Y 182.762,Z 432.368,A -85,B 0,C 180,E1 -23166.587,E2 -23166.587} C_VEL
LIN {X 0,Y 188.726,Z 421.485,A -85,B 0,C 180,E1 -23169.969,E2 -23169.969} C_VEL
LIN {X 0,Y 194.397,Z 410.288,A -85,B 0,C 180,E1 -23172.677,E2 -23172.677} C_VEL
LIN {X 0,Y 200.329,Z 397.483,A -85,B 0,C 180,E1 -23175.074,E2 -23175.074} C_VEL
LIN {X 0,Y 205.327,Z 384.529,A -85,B 0,C 180,E1 -23177.024,E2 -23177.024} C_VEL
LIN {X 0,Y 209.756,Z 371.271,A -85,B 0,C 180,E1 -23178.564,E2 -23178.564} C_VEL
LIN {X 0,Y 213.858,Z 356.764,A -85,B 0,C 180,E1 -23179.824,E2 -23179.824} C_VEL
LIN {X 0,Y 217.126,Z 341.717,A -85,B 0,C 180,E1 -23180.789,E2 -23180.789} C_VEL
LIN {X 0,Y 219.502,Z 325.845,A -85,B 0,C 180,E1 -23181.495,E2 -23181.495} C_VEL
LIN {X 0,Y 222.876,Z 283.891,A -85,B 0,C 180,E1 -23182.642,E2 -23182.642} C_VEL
LIN {X 0,Y 225.033,Z 252.901,A -85,B 0,C 180,E1 -23183.526,E2 -23183.526} C_VEL
LIN {X 0,Y 220.202,Z 241.145,A -85,B 0,C 180,E1 -23185.909,E2 -23185.909} C_VEL
LIN {X 0,Y 214.947,Z 229.886,A -85,B 0,C 180,E1 -23188.717,E2 -23188.717} C_VEL
LIN {X 0,Y 210.447,Z 221.12,A -85,B 0,C 180,E1 -23191.379,E2 -23191.379} C_VEL
LIN {X 0,Y 207.789,Z 216.596,A -85,B 0,C 180,E1 -23193.073,E2 -23193.073} C_VEL
LIN {X 0,Y 205.115,Z 212.706,A -85,B 0,C 180,E1 -23194.878,E2 -23194.878} C_VEL
LIN {X 0,Y 202.557,Z 209.095,A -85,B 0,C 180,E1 -23196.765,E2 -23196.765} C_VEL
LIN {X 0,Y 199.852,Z 205.308,A -85,B 0,C 180,E1 -23198.987,E2 -23198.987} C_VEL
LIN {X 0,Y 196.872,Z 201.25,A -85,B 0,C 180,E1 -23201.799,E2 -23201.799} C_VEL
LIN {X 0,Y 193.87,Z 197.739,A -85,B 0,C 180,E1 -23205.164,E2 -23205.164} C_VEL
LIN {X 0,Y 192.716,Z 195.629,A -85,B 0,C 180,E1 -23206.825,E2 -23206.825} C_VEL
LIN {X 0,Y 190.227,Z 193.375,A -85,B 0,C 180,E1 -23210.966,E2 -23210.966} C_VEL
LIN {X 0,Y 189.021,Z 190.256,A -85,B 0,C 180,E1 -23214.667,E2 -23214.667} C_VEL
LIN {X 0,Y 188.202,Z 189.717,A -85,B 0,C 180,E1 -23220,E2 -23220} C_VEL
LIN {X 0,Y 189.04,Z 190.355,A -85,B 0,C 180,E1 -23225.868,E2 -23225.868} C_VEL
LIN {X 0,Y 190.515,Z 193.842,A -85,B 0,C 180,E1 -23230.092,E2 -23230.092} C_VEL
LIN {X 0,Y 192.951,Z 196.025,A -85,B 0,C 180,E1 -23233.964,E2 -23233.964} C_VEL
LIN {X 0,Y 195.066,Z 199.48,A -85,B 0,C 180,E1 -23236.752,E2 -23236.752} C_VEL
LIN {X 0,Y 196.836,Z 201.25,A -85,B 0,C 180,E1 -23238.609,E2 -23238.609} C_VEL
LIN {X 0,Y 199.508,Z 205.005,A -85,B 0,C 180,E1 -23241.166,E2 -23241.166} C_VEL
LIN {X 0,Y 200.634,Z 206.384,A -85,B 0,C 180,E1 -23242.121,E2 -23242.121} C_VEL
LIN {X 0,Y 203.918,Z 211.027,A -85,B 0,C 180,E1 -23244.702,E2 -23244.702} C_VEL
LIN {X 0,Y 207.622,Z 216.384,A -85,B 0,C 180,E1 -23247.26,E2 -23247.26} C_VEL
LIN {X 0,Y 211.748,Z 222.555,A -85,B 0,C 180,E1 -23249.79,E2 -23249.79} C_VEL
LIN {X 0,Y 217.837,Z 232.722,A -85,B 0,C 180,E1 -23253.11,E2 -23253.11} C_VEL
LIN {X 0,Y 223.596,Z 243.316,A -85,B 0,C 180,E1 -23255.902,E2 -23255.902} C_VEL
LIN {X 0,Y 225.407,Z 246.899,A -85,B 0,C 180,E1 -23256.727,E2 -23256.727} C_VEL
LIN {X 0,Y 222.563,Z 285.654,A -85,B 0,C 180,E1 -23257.783,E2 -23257.783} C_VEL
LIN {X 0,Y 220.01,Z 318.324,A -85,B 0,C 180,E1 -23258.728,E2 -23258.728} C_VEL
LIN {X 0,Y 217.744,Z 333.627,A -85,B 0,C 180,E1 -23259.41,E2 -23259.41} C_VEL
LIN {X 0,Y 214.684,Z 348.723,A -85,B 0,C 180,E1 -23260.436,E2 -23260.436} C_VEL
LIN {X 0,Y 211.123,Z 362.454,A -85,B 0,C 180,E1 -23261.699,E2 -23261.699} C_VEL
LIN {X 0,Y 206.716,Z 376.452,A -85,B 0,C 180,E1 -23263.388,E2 -23263.388} C_VEL
LIN {X 0,Y 201.44,Z 389.897,A -85,B 0,C 180,E1 -23265.401,E2 -23265.401} C_VEL
LIN {X 0,Y 196.019,Z 402.097,A -85,B 0,C 180,E1 -23267.759,E2 -23267.759} C_VEL
LIN {X 0,Y 190.393,Z 413.215,A -85,B 0,C 180,E1 -23270.45,E2 -23270.45} C_VEL
LIN {X 0,Y 186.164,Z 421.078,A -85,B 0,C 180,E1 -23272.841,E2 -23272.841} C_VEL
LIN {X 0,Y 181.454,Z 429.293,A -85,B 0,C 180,E1 -23275.833,E2 -23275.833} C_VEL
LIN {X 0,Y 176.545,Z 437.367,A -85,B 0,C 180,E1 -23279.499,E2 -23279.499} C_VEL
LIN {X 0,Y 171.529,Z 445.149,A -85,B 0,C 180,E1 -23284.073,E2 -23284.073} C_VEL
LIN {X 0,Y 167.61,Z 451.497,A -85,B 0,C 180,E1 -23289.12,E2 -23289.12} C_VEL
LIN {X 0,Y 165.415,Z 454.934,A -85,B 0,C 180,E1 -23292.698,E2 -23292.698} C_VEL
LIN {X 0,Y 163.514,Z 458.402,A -85,B 0,C 180,E1 -23297.59,E2 -23297.59} C_VEL
LIN {X 0,Y 162.376,Z 460.69,A -85,B 0,C 180,E1 -23302.539,E2 -23302.539} C_VEL
LIN {X 0,Y 161.926,Z 461.852,A -85,B 0,C 180,E1 -23307.513,E2 -23307.513} C_VEL
LIN {X 0,Y 161.939,Z 462.005,A -85,B 0,C 180,E1 -23310,E2 -23310} C_VEL
LIN {X 0,Y 162.067,Z 461.444,A -85,B 0,C 180,E1 -23314.976,E2 -23314.976} C_VEL
LIN {X 0,Y 162.828,Z 459.77,A -85,B 0,C 180,E1 -23319.942,E2 -23319.942} C_VEL
LIN {X 0,Y 164.294,Z 456.943,A -85,B 0,C 180,E1 -23324.872,E2 -23324.872} C_VEL
LIN {X 0,Y 166.812,Z 452.886,A -85,B 0,C 180,E1 -23329.697,E2 -23329.697} C_VEL
LIN {X 0,Y 170.144,Z 447.506,A -85,B 0,C 180,E1 -23334.398,E2 -23334.398} C_VEL
LIN {X 0,Y 174.54,Z 440.641,A -85,B 0,C 180,E1 -23338.894,E2 -23338.894} C_VEL
LIN {X 0,Y 179.87,Z 432.067,A -85,B 0,C 180,E1 -23343.163,E2 -23343.163} C_VEL
LIN {X 0,Y 185.332,Z 422.941,A -85,B 0,C 180,E1 -23346.674,E2 -23346.674} C_VEL
LIN {X 0,Y 190.285,Z 413.653,A -85,B 0,C 180,E1 -23349.577,E2 -23349.577} C_VEL
LIN {X 0,Y 196.401,Z 401.611,A -85,B 0,C 180,E1 -23352.487,E2 -23352.487} C_VEL
LIN {X 0,Y 201.836,Z 389.313,A -85,B 0,C 180,E1 -23354.839,E2 -23354.839} C_VEL
LIN {X 0,Y 206.953,Z 376.067,A -85,B 0,C 180,E1 -23356.82,E2 -23356.82} C_VEL
LIN {X 0,Y 211.051,Z 363.098,A -85,B 0,C 180,E1 -23358.382,E2 -23358.382} C_VEL
LIN {X 0,Y 214.861,Z 348.754,A -85,B 0,C 180,E1 -23359.689,E2 -23359.689} C_VEL
LIN {X 0,Y 218.1,Z 332.924,A -85,B 0,C 180,E1 -23360.745,E2 -23360.745} C_VEL
LIN {X 0,Y 220.326,Z 317.494,A -85,B 0,C 180,E1 -23361.423,E2 -23361.423} C_VEL
LIN {X 0,Y 225.638,Z 247.182,A -85,B 0,C 180,E1 -23363.372,E2 -23363.372} C_VEL
LIN {X 0,Y 220.089,Z 236.609,A -85,B 0,C 180,E1 -23365.977,E2 -23365.977} C_VEL
LIN {X 0,Y 214.699,Z 227.3,A -85,B 0,C 180,E1 -23368.772,E2 -23368.772} C_VEL
LIN {X 0,Y 210.33,Z 220.336,A -85,B 0,C 180,E1 -23371.293,E2 -23371.293} C_VEL
LIN {X 0,Y 206.212,Z 214.058,A -85,B 0,C 180,E1 -23373.961,E2 -23373.961} C_VEL
LIN {X 0,Y 202.709,Z 209.261,A -85,B 0,C 180,E1 -23376.502,E2 -23376.502} C_VEL
LIN {X 0,Y 199.845,Z 205.32,A -85,B 0,C 180,E1 -23378.871,E2 -23378.871} C_VEL
LIN {X 0,Y 197.156,Z 201.702,A -85,B 0,C 180,E1 -23381.422,E2 -23381.422} C_VEL
LIN {X 0,Y 196.336,Z 200.599,A -85,B 0,C 180,E1 -23382.286,E2 -23382.286} C_VEL
LIN {X 0,Y 193.943,Z 197.866,A -85,B 0,C 180,E1 -23385.066,E2 -23385.066} C_VEL
LIN {X 0,Y 192.756,Z 195.632,A -85,B 0,C 180,E1 -23386.828,E2 -23386.828} C_VEL
LIN {X 0,Y 190.352,Z 193.461,A -85,B 0,C 180,E1 -23390.972,E2 -23390.972} C_VEL
LIN {X 0,Y 189.09,Z 190.185,A -85,B 0,C 180,E1 -23395.245,E2 -23395.245} C_VEL
LIN {X 0,Y 188.533,Z 189.811,A -85,B 0,C 180,E1 -23400,E2 -23400} C_VEL
LIN {X 0,Y 189.11,Z 190.29,A -85,B 0,C 180,E1 -23404.529,E2 -23404.529} C_VEL
LIN {X 0,Y 190.834,Z 194.111,A -85,B 0,C 180,E1 -23409.706,E2 -23409.706} C_VEL
LIN {X 0,Y 193.047,Z 196.017,A -85,B 0,C 180,E1 -23413.252,E2 -23413.252} C_VEL
LIN {X 0,Y 195.252,Z 199.565,A -85,B 0,C 180,E1 -23416.198,E2 -23416.198} C_VEL
LIN {X 0,Y 196.892,Z 201.198,A -85,B 0,C 180,E1 -23417.939,E2 -23417.939} C_VEL
LIN {X 0,Y 199.653,Z 205.058,A -85,B 0,C 180,E1 -23420.61,E2 -23420.61} C_VEL
LIN {X 0,Y 200.971,Z 206.823,A -85,B 0,C 180,E1 -23421.744,E2 -23421.744} C_VEL
LIN {X 0,Y 204.146,Z 211.258,A -85,B 0,C 180,E1 -23424.234,E2 -23424.234} C_VEL
LIN {X 0,Y 207.946,Z 216.714,A -85,B 0,C 180,E1 -23426.857,E2 -23426.857} C_VEL
LIN {X 0,Y 210.855,Z 221.701,A -85,B 0,C 180,E1 -23428.714,E2 -23428.714} C_VEL
LIN {X 0,Y 215.217,Z 230.261,A -85,B 0,C 180,E1 -23431.293,E2 -23431.293} C_VEL
LIN {X 0,Y 220.391,Z 241.364,A -85,B 0,C 180,E1 -23434.062,E2 -23434.062} C_VEL
LIN {X 0,Y 224.779,Z 252.016,A -85,B 0,C 180,E1 -23436.238,E2 -23436.238} C_VEL
LIN {X 0,Y 225.192,Z 253.112,A -85,B 0,C 180,E1 -23436.437,E2 -23436.437} C_VEL
LIN {X 0,Y 222.634,Z 289.261,A -85,B 0,C 180,E1 -23437.455,E2 -23437.455} C_VEL
LIN {X 0,Y 220.316,Z 319.749,A -85,B 0,C 180,E1 -23438.283,E2 -23438.283} C_VEL
LIN {X 0,Y 219.776,Z 323.64,A -85,B 0,C 180,E1 -23438.343,E2 -23438.343} C_VEL
LIN {X 0,Y 217.667,Z 331.258,A -85,B 0,C 180,E1 -23438.242,E2 -23438.242} C_VEL
LIN {X 0,Y 212.804,Z 344.255,A -85,B 0,C 180,E1 -23437.985,E2 -23437.985} C_VEL
LIN {X 0,Y 211.142,Z 349.878,A -85,B 0,C 180,E1 -23438.187,E2 -23438.187} C_VEL
LIN {X 0,Y 207.531,Z 363.799,A -85,B 0,C 180,E1 -23439.226,E2 -23439.226} C_VEL
LIN {X 0,Y 203.388,Z 376.856,A -85,B 0,C 180,E1 -23440.517,E2 -23440.517} C_VEL
LIN {X 0,Y 198.002,Z 391.204,A -85,B 0,C 180,E1 -23442.407,E2 -23442.407} C_VEL
LIN {X 0,Y 192.393,Z 403.97,A -85,B 0,C 180,E1 -23444.575,E2 -23444.575} C_VEL
LIN {X 0,Y 186.225,Z 416.164,A -85,B 0,C 180,E1 -23447.21,E2 -23447.21} C_VEL
LIN {X 0,Y 180.557,Z 426.41,A -85,B 0,C 180,E1 -23450.04,E2 -23450.04} C_VEL
LIN {X 0,Y 174.626,Z 436.46,A -85,B 0,C 180,E1 -23453.602,E2 -23453.602} C_VEL
LIN {X 0,Y 169.495,Z 444.756,A -85,B 0,C 180,E1 -23457.382,E2 -23457.382} C_VEL
LIN {X 0,Y 164.296,Z 452.579,A -85,B 0,C 180,E1 -23461.93,E2 -23461.93} C_VEL
LIN {X 0,Y 160.055,Z 459.35,A -85,B 0,C 180,E1 -23467.235,E2 -23467.235} C_VEL
LIN {X 0,Y 157.445,Z 463.647,A -85,B 0,C 180,E1 -23471.792,E2 -23471.792} C_VEL
LIN {X 0,Y 155.571,Z 467.192,A -85,B 0,C 180,E1 -23476.945,E2 -23476.945} C_VEL
LIN {X 0,Y 154.74,Z 469.533,A -85,B 0,C 180,E1 -23482.169,E2 -23482.169} C_VEL
LIN {X 0,Y 154.662,Z 470.716,A -85,B 0,C 180,E1 -23487.395,E2 -23487.395} C_VEL
LIN {X 0,Y 154.793,Z 470.874,A -85,B 0,C 180,E1 -23490,E2 -23490} C_VEL
LIN {X 0,Y 154.62,Z 470.25,A -85,B 0,C 180,E1 -23495.216,E2 -23495.216} C_VEL
LIN {X 0,Y 155.039,Z 468.469,A -85,B 0,C 180,E1 -23500.447,E2 -23500.447} C_VEL
LIN {X 0,Y 156.334,Z 465.514,A -85,B 0,C 180,E1 -23505.648,E2 -23505.648} C_VEL
LIN {X 0,Y 158.7,Z 461.321,A -85,B 0,C 180,E1 -23510.749,E2 -23510.749} C_VEL
LIN {X 0,Y 162.157,Z 455.779,A -85,B 0,C 180,E1 -23515.684,E2 -23515.684} C_VEL
LIN {X 0,Y 166.658,Z 448.74,A -85,B 0,C 180,E1 -23520.401,E2 -23520.401} C_VEL
LIN {X 0,Y 171.57,Z 441.225,A -85,B 0,C 180,E1 -23524.28,E2 -23524.28} C_VEL
LIN {X 0,Y 177.048,Z 432.164,A -85,B 0,C 180,E1 -23527.972,E2 -23527.972} C_VEL
LIN {X 0,Y 183.31,Z 421.283,A -85,B 0,C 180,E1 -23531.404,E2 -23531.404} C_VEL
LIN {X 0,Y 189.235,Z 410.086,A -85,B 0,C 180,E1 -23534.136,E2 -23534.136} C_VEL
LIN {X 0,Y 195.278,Z 397.469,A -85,B 0,C 180,E1 -23536.522,E2 -23536.522} C_VEL
LIN {X 0,Y 200.541,Z 384.326,A -85,B 0,C 180,E1 -23538.512,E2 -23538.512} C_VEL
LIN {X 0,Y 205.124,Z 371.066,A -85,B 0,C 180,E1 -23540.051,E2 -23540.051} C_VEL
LIN {X 0,Y 209.344,Z 356.558,A -85,B 0,C 180,E1 -23541.31,E2 -23541.31} C_VEL
LIN {X 0,Y 212.711,Z 341.508,A -85,B 0,C 180,E1 -23542.27,E2 -23542.27} C_VEL
LIN {X 0,Y 215.026,Z 326.488,A -85,B 0,C 180,E1 -23542.948,E2 -23542.948} C_VEL
LIN {X 0,Y 217.04,Z 303.689,A -85,B 0,C 180,E1 -23543.603,E2 -23543.603} C_VEL
LIN {X 0,Y 220.707,Z 255.716,A -85,B 0,C 180,E1 -23544.905,E2 -23544.905} C_VEL
LIN {X 0,Y 216.069,Z 244.191,A -85,B 0,C 180,E1 -23547.366,E2 -23547.366} C_VEL
LIN {X 0,Y 210.901,Z 232.942,A -85,B 0,C 180,E1 -23550.354,E2 -23550.354} C_VEL
LIN {X 0,Y 206.268,Z 223.865,A -85,B 0,C 180,E1 -23553.355,E2 -23553.355} C_VEL
LIN {X 0,Y 203.302,Z 219.372,A -85,B 0,C 180,E1 -23555.424,E2 -23555.424} C_VEL
LIN {X 0,Y 200.641,Z 215.479,A -85,B 0,C 180,E1 -23557.473,E2 -23557.473} C_VEL
LIN {X 0,Y 198.001,Z 211.688,A -85,B 0,C 180,E1 -23559.753,E2 -23559.753} C_VEL
LIN {X 0,Y 194.82,Z 207.279,A -85,B 0,C 180,E1 -23562.956,E2 -23562.956} C_VEL
LIN {X 0,Y 192.422,Z 204.277,A -85,B 0,C 180,E1 -23565.863,E2 -23565.863} C_VEL
LIN {X 0,Y 191.494,Z 202.503,A -85,B 0,C 180,E1 -23567.279,E2 -23567.279} C_VEL
LIN {X 0,Y 189.123,Z 200.201,A -85,B 0,C 180,E1 -23571.452,E2 -23571.452} C_VEL
LIN {X 0,Y 188.008,Z 197.211,A -85,B 0,C 180,E1 -23575.176,E2 -23575.176} C_VEL
LIN {X 0,Y 187.336,Z 196.766,A -85,B 0,C 180,E1 -23580,E2 -23580} C_VEL
LIN {X 0,Y 188.086,Z 197.468,A -85,B 0,C 180,E1 -23585.629,E2 -23585.629} C_VEL
LIN {X 0,Y 189.65,Z 200.995,A -85,B 0,C 180,E1 -23590.138,E2 -23590.138} C_VEL
LIN {X 0,Y 191.639,Z 202.739,A -85,B 0,C 180,E1 -23593.386,E2 -23593.386} C_VEL
LIN {X 0,Y 193.609,Z 206.12,A -85,B 0,C 180,E1 -23596.136,E2 -23596.136} C_VEL
LIN {X 0,Y 195.335,Z 207.978,A -85,B 0,C 180,E1 -23598.045,E2 -23598.045} C_VEL
LIN {X 0,Y 198.101,Z 211.847,A -85,B 0,C 180,E1 -23600.78,E2 -23600.78} C_VEL
LIN {X 0,Y 201.929,Z 217.37,A -85,B 0,C 180,E1 -23603.986,E2 -23603.986} C_VEL
LIN {X 0,Y 205.377,Z 222.493,A -85,B 0,C 180,E1 -23606.483,E2 -23606.483} C_VEL
LIN {X 0,Y 209.861,Z 229.558,A -85,B 0,C 180,E1 -23609.354,E2 -23609.354} C_VEL
LIN {X 0,Y 215.274,Z 238.974,A -85,B 0,C 180,E1 -23612.425,E2 -23612.425} C_VEL
LIN {X 0,Y 220.394,Z 248.724,A -85,B 0,C 180,E1 -23615.029,E2 -23615.029} C_VEL
LIN {X 0,Y 221.017,Z 249.954,A -85,B 0,C 180,E1 -23615.329,E2 -23615.329} C_VEL
LIN {X 0,Y 218.299,Z 285.741,A -85,B 0,C 180,E1 -23616.308,E2 -23616.308} C_VEL
LIN {X 0,Y 215.657,Z 318.432,A -85,B 0,C 180,E1 -23617.253,E2 -23617.253} C_VEL
LIN {X 0,Y 213.314,Z 333.836,A -85,B 0,C 180,E1 -23617.939,E2 -23617.939} C_VEL
LIN {X 0,Y 210.15,Z 348.929,A -85,B 0,C 180,E1 -23618.964,E2 -23618.964} C_VEL
LIN {X 0,Y 206.306,Z 363.181,A -85,B 0,C 180,E1 -23620.285,E2 -23620.285} C_VEL
LIN {X 0,Y 201.908,Z 376.655,A -85,B 0,C 180,E1 -23621.925,E2 -23621.925} C_VEL
LIN {X 0,Y 196.454,Z 390.1,A -85,B 0,C 180,E1 -23623.949,E2 -23623.949} C_VEL
LIN {X 0,Y 191.33,Z 401.263,A -85,B 0,C 180,E1 -23626.106,E2 -23626.106} C_VEL
LIN {X 0,Y 185.915,Z 411.65,A -85,B 0,C 180,E1 -23628.583,E2 -23628.583} C_VEL
LIN {X 0,Y 181.172,Z 420.073,A -85,B 0,C 180,E1 -23631.052,E2 -23631.052} C_VEL
LIN {X 0,Y 176.422,Z 428.233,A -85,B 0,C 180,E1 -23634.014,E2 -23634.014} C_VEL
LIN {X 0,Y 171.121,Z 436.484,A -85,B 0,C 180,E1 -23637.73,E2 -23637.73} C_VEL
LIN {X 0,Y 165.902,Z 444.231,A -85,B 0,C 180,E1 -23642.226,E2 -23642.226} C_VEL
LIN {X 0,Y 161.808,Z 450.386,A -85,B 0,C 180,E1 -23646.989,E2 -23646.989} C_VEL
LIN {X 0,Y 158.614,Z 455.135,A -85,B 0,C 180,E1 -23651.931,E2 -23651.931} C_VEL
LIN {X 0,Y 156.561,Z 458.602,A -85,B 0,C 180,E1 -23657.03,E2 -23657.03} C_VEL
LIN {X 0,Y 155.329,Z 460.889,A -85,B 0,C 180,E1 -23662.199,E2 -23662.199} C_VEL
LIN {X 0,Y 154.845,Z 462.05,A -85,B 0,C 180,E1 -23667.399,E2 -23667.399} C_VEL
LIN {X 0,Y 154.853,Z 462.204,A -85,B 0,C 180,E1 -23670,E2 -23670} C_VEL
LIN {X 0,Y 155.005,Z 461.642,A -85,B 0,C 180,E1 -23675.203,E2 -23675.203} C_VEL
LIN {X 0,Y 155.818,Z 459.969,A -85,B 0,C 180,E1 -23680.394,E2 -23680.394} C_VEL
LIN {X 0,Y 157.417,Z 457.142,A -85,B 0,C 180,E1 -23685.538,E2 -23685.538} C_VEL
LIN {X 0,Y 160.098,Z 453.085,A -85,B 0,C 180,E1 -23690.56,E2 -23690.56} C_VEL
LIN {X 0,Y 163.633,Z 447.706,A -85,B 0,C 180,E1 -23695.436,E2 -23695.436} C_VEL
LIN {X 0,Y 168.322,Z 440.84,A -85,B 0,C 180,E1 -23700.069,E2 -23700.069} C_VEL
LIN {X 0,Y 173.937,Z 432.264,A -85,B 0,C 180,E1 -23704.449,E2 -23704.449} C_VEL
LIN {X 0,Y 179.665,Z 423.139,A -85,B 0,C 180,E1 -23708.032,E2 -23708.032} C_VEL
LIN {X 0,Y 184.854,Z 413.85,A -85,B 0,C 180,E1 -23710.983,E2 -23710.983} C_VEL
LIN {X 0,Y 191.207,Z 401.807,A -85,B 0,C 180,E1 -23713.93,E2 -23713.93} C_VEL
LIN {X 0,Y 196.866,Z 389.508,A -85,B 0,C 180,E1 -23716.296,E2 -23716.296} C_VEL
LIN {X 0,Y 202.056,Z 376.565,A -85,B 0,C 180,E1 -23718.245,E2 -23718.245} C_VEL
LIN {X 0,Y 206.415,Z 363.29,A -85,B 0,C 180,E1 -23719.852,E2 -23719.852} C_VEL
LIN {X 0,Y 210.35,Z 348.944,A -85,B 0,C 180,E1 -23721.16,E2 -23721.16} C_VEL
LIN {X 0,Y 213.552,Z 333.847,A -85,B 0,C 180,E1 -23722.171,E2 -23722.171} C_VEL
LIN {X 0,Y 215.827,Z 318.676,A -85,B 0,C 180,E1 -23722.863,E2 -23722.863} C_VEL
LIN {X 0,Y 219.143,Z 277.724,A -85,B 0,C 180,E1 -23724.025,E2 -23724.025} C_VEL
LIN {X 0,Y 221.243,Z 250.221,A -85,B 0,C 180,E1 -23724.773,E2 -23724.773} C_VEL
LIN {X 0,Y 215.747,Z 239.568,A -85,B 0,C 180,E1 -23727.556,E2 -23727.556} C_VEL
LIN {X 0,Y 210.106,Z 229.812,A -85,B 0,C 180,E1 -23730.746,E2 -23730.746} C_VEL
LIN {X 0,Y 205.625,Z 222.736,A -85,B 0,C 180,E1 -23733.62,E2 -23733.62} C_VEL
LIN {X 0,Y 201.24,Z 216.158,A -85,B 0,C 180,E1 -23736.865,E2 -23736.865} C_VEL
LIN {X 0,Y 198.162,Z 211.889,A -85,B 0,C 180,E1 -23739.499,E2 -23739.499} C_VEL
LIN {X 0,Y 195.409,Z 207.958,A -85,B 0,C 180,E1 -23742.267,E2 -23742.267} C_VEL
LIN {X 0,Y 192.332,Z 204.092,A -85,B 0,C 180,E1 -23746.024,E2 -23746.024} C_VEL
LIN {X 0,Y 191.542,Z 202.531,A -85,B 0,C 180,E1 -23747.282,E2 -23747.282} C_VEL
LIN {X 0,Y 189.262,Z 200.274,A -85,B 0,C 180,E1 -23751.458,E2 -23751.458} C_VEL
LIN {X 0,Y 188.107,Z 197.213,A -85,B 0,C 180,E1 -23755.714,E2 -23755.714} C_VEL
LIN {X 0,Y 187.669,Z 196.849,A -85,B 0,C 180,E1 -23760,E2 -23760} C_VEL
LIN {X 0,Y 188.172,Z 197.379,A -85,B 0,C 180,E1 -23764.284,E2 -23764.284} C_VEL
LIN {X 0,Y 190.072,Z 201.382,A -85,B 0,C 180,E1 -23769.952,E2 -23769.952} C_VEL
LIN {X 0,Y 191.759,Z 202.807,A -85,B 0,C 180,E1 -23772.703,E2 -23772.703} C_VEL
LIN {X 0,Y 194.175,Z 206.61,A -85,B 0,C 180,E1 -23776.02,E2 -23776.02} C_VEL
LIN {X 0,Y 195.422,Z 207.985,A -85,B 0,C 180,E1 -23777.4,E2 -23777.4} C_VEL
LIN {X 0,Y 198.384,Z 212.056,A -85,B 0,C 180,E1 -23780.342,E2 -23780.342} C_VEL
LIN {X 0,Y 202.224,Z 217.697,A -85,B 0,C 180,E1 -23783.568,E2 -23783.568} C_VEL
LIN {X 0,Y 206.224,Z 223.605,A -85,B 0,C 180,E1 -23786.434,E2 -23786.434} C_VEL
LIN {X 0,Y 210.839,Z 232.617,A -85,B 0,C 180,E1 -23789.451,E2 -23789.451} C_VEL
LIN {X 0,Y 215.734,Z 243.226,A -85,B 0,C 180,E1 -23792.312,E2 -23792.312} C_VEL
LIN {X 0,Y 220.32,Z 254.32,A -85,B 0,C 180,E1 -23794.764,E2 -23794.764} C_VEL
LIN {X 0,Y 220.918,Z 255.904,A -85,B 0,C 180,E1 -23795.072,E2 -23795.072} C_VEL
LIN {X 0,Y 215.449,Z 325.092,A -85,B 0,C 180,E1 -23796.977,E2 -23796.977} C_VEL
LIN {X 0,Y 213.071,Z 340.804,A -85,B 0,C 180,E1 -23797.662,E2 -23797.662} C_VEL
LIN {X 0,Y 211.142,Z 349.878,A -85,B 0,C 180,E1 -23798.187,E2 -23798.187} C_VEL
LIN {X 0,Y 209.372,Z 355.472,A -85,B 0,C 180,E1 -23798.415,E2 -23798.415} C_VEL
LIN {X 0,Y 201.368,Z 371.397,A -85,B 0,C 180,E1 -23798.636,E2 -23798.636} C_VEL
LIN {X 0,Y 198.899,Z 376.629,A -85,B 0,C 180,E1 -23798.972,E2 -23798.972} C_VEL
LIN {X 0,Y 198.216,Z 378.344,A -85,B 0,C 180,E1 -23799.159,E2 -23799.159} C_VEL
LIN {X 0,Y 192.854,Z 391.94,A -85,B 0,C 180,E1 -23800.992,E2 -23800.992} C_VEL
LIN {X 0,Y 187.462,Z 403.774,A -85,B 0,C 180,E1 -23803.024,E2 -23803.024} C_VEL
LIN {X 0,Y 181.043,Z 415.967,A -85,B 0,C 180,E1 -23805.673,E2 -23805.673} C_VEL
LIN {X 0,Y 175.14,Z 426.212,A -85,B 0,C 180,E1 -23808.538,E2 -23808.538} C_VEL
LIN {X 0,Y 168.801,Z 436.411,A -85,B 0,C 180,E1 -23812.217,E2 -23812.217} C_VEL
LIN {X 0,Y 162.783,Z 445.638,A -85,B 0,C 180,E1 -23816.6,E2 -23816.6} C_VEL
LIN {X 0,Y 157.997,Z 452.38,A -85,B 0,C 180,E1 -23820.705,E2 -23820.705} C_VEL
LIN {X 0,Y 153.768,Z 458.616,A -85,B 0,C 180,E1 -23825.71,E2 -23825.71} C_VEL
LIN {X 0,Y 150.636,Z 463.446,A -85,B 0,C 180,E1 -23830.938,E2 -23830.938} C_VEL
LIN {X 0,Y 148.595,Z 466.992,A -85,B 0,C 180,E1 -23836.321,E2 -23836.321} C_VEL
LIN {X 0,Y 147.689,Z 469.334,A -85,B 0,C 180,E1 -23841.792,E2 -23841.792} C_VEL
LIN {X 0,Y 147.564,Z 470.517,A -85,B 0,C 180,E1 -23847.27,E2 -23847.27} C_VEL
LIN {X 0,Y 147.716,Z 470.676,A -85,B 0,C 180,E1 -23850,E2 -23850} C_VEL
LIN {X 0,Y 147.533,Z 470.051,A -85,B 0,C 180,E1 -23855.467,E2 -23855.467} C_VEL
LIN {X 0,Y 148.014,Z 468.269,A -85,B 0,C 180,E1 -23860.949,E2 -23860.949} C_VEL
LIN {X 0,Y 149.46,Z 465.313,A -85,B 0,C 180,E1 -23866.388,E2 -23866.388} C_VEL
LIN {X 0,Y 152.003,Z 461.118,A -85,B 0,C 180,E1 -23871.709,E2 -23871.709} C_VEL
LIN {X 0,Y 155.725,Z 455.577,A -85,B 0,C 180,E1 -23876.828,E2 -23876.828} C_VEL
LIN {X 0,Y 160.515,Z 448.538,A -85,B 0,C 180,E1 -23881.696,E2 -23881.696} C_VEL
LIN {X 0,Y 165.655,Z 441.021,A -85,B 0,C 180,E1 -23885.687,E2 -23885.687} C_VEL
LIN {X 0,Y 171.445,Z 431.961,A -85,B 0,C 180,E1 -23889.449,E2 -23889.449} C_VEL
LIN {X 0,Y 178.011,Z 421.08,A -85,B 0,C 180,E1 -23892.925,E2 -23892.925} C_VEL
LIN {X 0,Y 184.198,Z 409.884,A -85,B 0,C 180,E1 -23895.676,E2 -23895.676} C_VEL
LIN {X 0,Y 190.34,Z 397.49,A -85,B 0,C 180,E1 -23898.038,E2 -23898.038} C_VEL
LIN {X 0,Y 195.889,Z 384.121,A -85,B 0,C 180,E1 -23900.075,E2 -23900.075} C_VEL
LIN {X 0,Y 200.643,Z 370.862,A -85,B 0,C 180,E1 -23901.604,E2 -23901.604} C_VEL
LIN {X 0,Y 204.663,Z 357.481,A -85,B 0,C 180,E1 -23902.773,E2 -23902.773} C_VEL
LIN {X 0,Y 208.292,Z 342.064,A -85,B 0,C 180,E1 -23903.767,E2 -23903.767} C_VEL
LIN {X 0,Y 210.706,Z 327.159,A -85,B 0,C 180,E1 -23904.453,E2 -23904.453} C_VEL
LIN {X 0,Y 212.801,Z 304.953,A -85,B 0,C 180,E1 -23905.095,E2 -23905.095} C_VEL
LIN {X 0,Y 216.474,Z 258.408,A -85,B 0,C 180,E1 -23906.362,E2 -23906.362} C_VEL
LIN {X 0,Y 211.958,Z 247.018,A -85,B 0,C 180,E1 -23908.948,E2 -23908.948} C_VEL
LIN {X 0,Y 207.207,Z 236.435,A -85,B 0,C 180,E1 -23911.933,E2 -23911.933} C_VEL
LIN {X 0,Y 203.448,Z 228.999,A -85,B 0,C 180,E1 -23914.555,E2 -23914.555} C_VEL
LIN {X 0,Y 199.171,Z 222.385,A -85,B 0,C 180,E1 -23917.855,E2 -23917.855} C_VEL
LIN {X 0,Y 196.173,Z 218.056,A -85,B 0,C 180,E1 -23920.545,E2 -23920.545} C_VEL
LIN {X 0,Y 193.282,Z 213.907,A -85,B 0,C 180,E1 -23923.623,E2 -23923.623} C_VEL
LIN {X 0,Y 190.986,Z 210.751,A -85,B 0,C 180,E1 -23926.602,E2 -23926.602} C_VEL
LIN {X 0,Y 190.281,Z 209.395,A -85,B 0,C 180,E1 -23927.739,E2 -23927.739} C_VEL
LIN {X 0,Y 188.033,Z 207.027,A -85,B 0,C 180,E1 -23931.943,E2 -23931.943} C_VEL
LIN {X 0,Y 187.074,Z 204.226,A -85,B 0,C 180,E1 -23935.421,E2 -23935.421} C_VEL
LIN {X 0,Y 186.471,Z 203.814,A -85,B 0,C 180,E1 -23940,E2 -23940} C_VEL
LIN {X 0,Y 187.115,Z 204.432,A -85,B 0,C 180,E1 -23945.253,E2 -23945.253} C_VEL
LIN {X 0,Y 188.685,Z 208.048,A -85,B 0,C 180,E1 -23949.988,E2 -23949.988} C_VEL
LIN {X 0,Y 190.417,Z 209.664,A -85,B 0,C 180,E1 -23952.93,E2 -23952.93} C_VEL
LIN {X 0,Y 192.482,Z 213.136,A -85,B 0,C 180,E1 -23955.893,E2 -23955.893} C_VEL
LIN {X 0,Y 193.857,Z 214.677,A -85,B 0,C 180,E1 -23957.471,E2 -23957.471} C_VEL
LIN {X 0,Y 196.571,Z 218.525,A -85,B 0,C 180,E1 -23960.265,E2 -23960.265} C_VEL
LIN {X 0,Y 200.23,Z 224.108,A -85,B 0,C 180,E1 -23963.464,E2 -23963.464} C_VEL
LIN {X 0,Y 203.494,Z 229.136,A -85,B 0,C 180,E1 -23965.922,E2 -23965.922} C_VEL
LIN {X 0,Y 207.739,Z 236.096,A -85,B 0,C 180,E1 -23968.754,E2 -23968.754} C_VEL
LIN {X 0,Y 213.186,Z 245.99,A -85,B 0,C 180,E1 -23971.966,E2 -23971.966} C_VEL
LIN {X 0,Y 216.746,Z 253.044,A -85,B 0,C 180,E1 -23973.871,E2 -23973.871} C_VEL
LIN {X 0,Y 214.576,Z 281.806,A -85,B 0,C 180,E1 -23974.693,E2 -23974.693} C_VEL
LIN {X 0,Y 211.452,Z 318.651,A -85,B 0,C 180,E1 -23975.729,E2 -23975.729} C_VEL
LIN {X 0,Y 209.035,Z 334.044,A -85,B 0,C 180,E1 -23976.408,E2 -23976.408} C_VEL
LIN {X 0,Y 205.761,Z 349.135,A -85,B 0,C 180,E1 -23977.427,E2 -23977.427} C_VEL
LIN {X 0,Y 202.043,Z 362.56,A -85,B 0,C 180,E1 -23978.655,E2 -23978.655} C_VEL
LIN {X 0,Y 197.24,Z 376.859,A -85,B 0,C 180,E1 -23980.392,E2 -23980.392} C_VEL
LIN {X 0,Y 192.131,Z 389.063,A -85,B 0,C 180,E1 -23982.206,E2 -23982.206} C_VEL
LIN {X 0,Y 186.771,Z 400.402,A -85,B 0,C 180,E1 -23984.361,E2 -23984.361} C_VEL
LIN {X 0,Y 180.64,Z 411.852,A -85,B 0,C 180,E1 -23987.089,E2 -23987.089} C_VEL
LIN {X 0,Y 174.975,Z 421.483,A -85,B 0,C 180,E1 -23990.01,E2 -23990.01} C_VEL
LIN {X 0,Y 169.852,Z 429.696,A -85,B 0,C 180,E1 -23993.132,E2 -23993.132} C_VEL
LIN {X 0,Y 164.391,Z 437.771,A -85,B 0,C 180,E1 -23996.97,E2 -23996.97} C_VEL
LIN {X 0,Y 159.621,Z 444.432,A -85,B 0,C 180,E1 -24001.032,E2 -24001.032} C_VEL
LIN {X 0,Y 155.242,Z 450.588,A -85,B 0,C 180,E1 -24005.956,E2 -24005.956} C_VEL
LIN {X 0,Y 151.846,Z 455.335,A -85,B 0,C 180,E1 -24011.096,E2 -24011.096} C_VEL
LIN {X 0,Y 149.635,Z 458.802,A -85,B 0,C 180,E1 -24016.418,E2 -24016.418} C_VEL
LIN {X 0,Y 148.278,Z 461.089,A -85,B 0,C 180,E1 -24021.825,E2 -24021.825} C_VEL
LIN {X 0,Y 147.756,Z 462.249,A -85,B 0,C 180,E1 -24027.274,E2 -24027.274} C_VEL
LIN {X 0,Y 147.766,Z 462.402,A -85,B 0,C 180,E1 -24030,E2 -24030} C_VEL
LIN {X 0,Y 147.937,Z 461.841,A -85,B 0,C 180,E1 -24035.452,E2 -24035.452} C_VEL
LIN {X 0,Y 148.832,Z 460.167,A -85,B 0,C 180,E1 -24040.888,E2 -24040.888} C_VEL
LIN {X 0,Y 150.57,Z 457.34,A -85,B 0,C 180,E1 -24046.264,E2 -24046.264} C_VEL
LIN {X 0,Y 153.431,Z 453.284,A -85,B 0,C 180,E1 -24051.497,E2 -24051.497} C_VEL
LIN {X 0,Y 157.383,Z 447.67,A -85,B 0,C 180,E1 -24056.733,E2 -24056.733} C_VEL
LIN {X 0,Y 162.198,Z 441.038,A -85,B 0,C 180,E1 -24061.33,E2 -24061.33} C_VEL
LIN {X 0,Y 168.106,Z 432.462,A -85,B 0,C 180,E1 -24065.824,E2 -24065.824} C_VEL
LIN {X 0,Y 174.099,Z 423.336,A -85,B 0,C 180,E1 -24069.479,E2 -24069.479} C_VEL
LIN {X 0,Y 179.536,Z 414.046,A -85,B 0,C 180,E1 -24072.474,E2 -24072.474} C_VEL
LIN {X 0,Y 186.136,Z 402.003,A -85,B 0,C 180,E1 -24075.453,E2 -24075.453} C_VEL
LIN {X 0,Y 192.035,Z 389.702,A -85,B 0,C 180,E1 -24077.826,E2 -24077.826} C_VEL
LIN {X 0,Y 197.287,Z 377.044,A -85,B 0,C 180,E1 -24079.743,E2 -24079.743} C_VEL
LIN {X 0,Y 201.553,Z 364.547,A -85,B 0,C 180,E1 -24081.278,E2 -24081.278} C_VEL
LIN {X 0,Y 205.676,Z 350.263,A -85,B 0,C 180,E1 -24082.605,E2 -24082.605} C_VEL
LIN {X 0,Y 208.959,Z 335.558,A -85,B 0,C 180,E1 -24083.62,E2 -24083.62} C_VEL
LIN {X 0,Y 211.377,Z 320.828,A -85,B 0,C 180,E1 -24084.309,E2 -24084.309} C_VEL
LIN {X 0,Y 213.387,Z 299.208,A -85,B 0,C 180,E1 -24084.968,E2 -24084.968} C_VEL
LIN {X 0,Y 217.043,Z 253.38,A -85,B 0,C 180,E1 -24086.201,E2 -24086.201} C_VEL
LIN {X 0,Y 211.446,Z 242.515,A -85,B 0,C 180,E1 -24089.258,E2 -24089.258} C_VEL
LIN {X 0,Y 206.022,Z 232.995,A -85,B 0,C 180,E1 -24092.62,E2 -24092.62} C_VEL
LIN {X 0,Y 201.543,Z 225.922,A -85,B 0,C 180,E1 -24095.812,E2 -24095.812} C_VEL
LIN {X 0,Y 198.867,Z 221.953,A -85,B 0,C 180,E1 -24097.979,E2 -24097.979} C_VEL
LIN {X 0,Y 196.373,Z 218.307,A -85,B 0,C 180,E1 -24100.259,E2 -24100.259} C_VEL
LIN {X 0,Y 193.469,Z 214.094,A -85,B 0,C 180,E1 -24103.377,E2 -24103.377} C_VEL
LIN {X 0,Y 190.957,Z 210.685,A -85,B 0,C 180,E1 -24106.701,E2 -24106.701} C_VEL
LIN {X 0,Y 190.424,Z 209.501,A -85,B 0,C 180,E1 -24107.612,E2 -24107.612} C_VEL
LIN {X 0,Y 188.234,Z 207.191,A -85,B 0,C 180,E1 -24111.816,E2 -24111.816} C_VEL
LIN {X 0,Y 187.236,Z 204.331,A -85,B 0,C 180,E1 -24115.694,E2 -24115.694} C_VEL
LIN {X 0,Y 186.803,Z 203.898,A -85,B 0,C 180,E1 -24120,E2 -24120} C_VEL
LIN {X 0,Y 187.241,Z 204.44,A -85,B 0,C 180,E1 -24124.035,E2 -24124.035} C_VEL
LIN {X 0,Y 189.104,Z 208.415,A -85,B 0,C 180,E1 -24129.795,E2 -24129.795} C_VEL
LIN {X 0,Y 190.584,Z 209.793,A -85,B 0,C 180,E1 -24132.309,E2 -24132.309} C_VEL
LIN {X 0,Y 192.992,Z 213.537,A -85,B 0,C 180,E1 -24135.714,E2 -24135.714} C_VEL
LIN {X 0,Y 194.073,Z 214.932,A -85,B 0,C 180,E1 -24136.971,E2 -24136.971} C_VEL
LIN {X 0,Y 197.422,Z 219.745,A -85,B 0,C 180,E1 -24140.377,E2 -24140.377} C_VEL
LIN {X 0,Y 200.548,Z 224.469,A -85,B 0,C 180,E1 -24143.065,E2 -24143.065} C_VEL
LIN {X 0,Y 203.911,Z 229.637,A -85,B 0,C 180,E1 -24145.588,E2 -24145.588} C_VEL
LIN {X 0,Y 207.993,Z 237.906,A -85,B 0,C 180,E1 -24148.418,E2 -24148.418} C_VEL
LIN {X 0,Y 212.632,Z 248.356,A -85,B 0,C 180,E1 -24151.302,E2 -24151.302} C_VEL
LIN {X 0,Y 216.669,Z 258.527,A -85,B 0,C 180,E1 -24153.603,E2 -24153.603} C_VEL
LIN {X 0,Y 211.269,Z 324.893,A -85,B 0,C 180,E1 -24155.442,E2 -24155.442} C_VEL
LIN {X 0,Y 208.793,Z 340.613,A -85,B 0,C 180,E1 -24156.114,E2 -24156.114} C_VEL
LIN {X 0,Y 205.327,Z 355.845,A -85,B 0,C 180,E1 -24157.065,E2 -24157.065} C_VEL
LIN {X 0,Y 201.241,Z 369.569,A -85,B 0,C 180,E1 -24158.207,E2 -24158.207} C_VEL
LIN {X 0,Y 198.216,Z 378.344,A -85,B 0,C 180,E1 -24159.159,E2 -24159.159} C_VEL
LIN {X 0,Y 195.872,Z 383.543,A -85,B 0,C 180,E1 -24159.656,E2 -24159.656} C_VEL
LIN {X 0,Y 186.154,Z 398.111,A -85,B 0,C 180,E1 -24160.652,E2 -24160.652} C_VEL
LIN {X 0,Y 183.138,Z 402.797,A -85,B 0,C 180,E1 -24161.261,E2 -24161.261} C_VEL
LIN {X 0,Y 182.277,Z 404.329,A -85,B 0,C 180,E1 -24161.54,E2 -24161.54} C_VEL
LIN {X 0,Y 176.001,Z 415.769,A -85,B 0,C 180,E1 -24164.047,E2 -24164.047} C_VEL
LIN {X 0,Y 169.841,Z 426.014,A -85,B 0,C 180,E1 -24166.939,E2 -24166.939} C_VEL
LIN {X 0,Y 163.316,Z 436.028,A -85,B 0,C 180,E1 -24170.598,E2 -24170.598} C_VEL
LIN {X 0,Y 157.631,Z 444.359,A -85,B 0,C 180,E1 -24174.577,E2 -24174.577} C_VEL
LIN {X 0,Y 151.788,Z 452.18,A -85,B 0,C 180,E1 -24179.381,E2 -24179.381} C_VEL
LIN {X 0,Y 147.253,Z 458.416,A -85,B 0,C 180,E1 -24184.561,E2 -24184.561} C_VEL
LIN {X 0,Y 143.871,Z 463.246,A -85,B 0,C 180,E1 -24190.004,E2 -24190.004} C_VEL
LIN {X 0,Y 141.642,Z 466.792,A -85,B 0,C 180,E1 -24195.635,E2 -24195.635} C_VEL
LIN {X 0,Y 140.629,Z 469.135,A -85,B 0,C 180,E1 -24201.377,E2 -24201.377} C_VEL
LIN {X 0,Y 140.48,Z 470.318,A -85,B 0,C 180,E1 -24207.132,E2 -24207.132} C_VEL
LIN {X 0,Y 140.568,Z 470.444,A -85,B 0,C 180,E1 -24210.644,E2 -24210.644} C_VEL
LIN {X 0,Y 140.441,Z 469.851,A -85,B 0,C 180,E1 -24215.744,E2 -24215.744} C_VEL
LIN {X 0,Y 141.011,Z 468.068,A -85,B 0,C 180,E1 -24221.499,E2 -24221.499} C_VEL
LIN {X 0,Y 142.615,Z 465.112,A -85,B 0,C 180,E1 -24227.198,E2 -24227.198} C_VEL
LIN {X 0,Y 145.343,Z 460.916,A -85,B 0,C 180,E1 -24232.758,E2 -24232.758} C_VEL
LIN {X 0,Y 149.353,Z 455.375,A -85,B 0,C 180,E1 -24238.071,E2 -24238.071} C_VEL
LIN {X 0,Y 154.478,Z 448.336,A -85,B 0,C 180,E1 -24243.089,E2 -24243.089} C_VEL
LIN {X 0,Y 159.875,Z 440.818,A -85,B 0,C 180,E1 -24247.189,E2 -24247.189} C_VEL
LIN {X 0,Y 165.967,Z 431.758,A -85,B 0,C 180,E1 -24251.023,E2 -24251.023} C_VEL
LIN {X 0,Y 172.858,Z 420.878,A -85,B 0,C 180,E1 -24254.535,E2 -24254.535} C_VEL
LIN {X 0,Y 179.297,Z 409.682,A -85,B 0,C 180,E1 -24257.303,E2 -24257.303} C_VEL
LIN {X 0,Y 185.869,Z 396.79,A -85,B 0,C 180,E1 -24259.767,E2 -24259.767} C_VEL
LIN {X 0,Y 191.394,Z 383.917,A -85,B 0,C 180,E1 -24261.711,E2 -24261.711} C_VEL
LIN {X 0,Y 196.312,Z 370.658,A -85,B 0,C 180,E1 -24263.229,E2 -24263.229} C_VEL
LIN {X 0,Y 200.441,Z 357.275,A -85,B 0,C 180,E1 -24264.392,E2 -24264.392} C_VEL
LIN {X 0,Y 204.014,Z 342.619,A -85,B 0,C 180,E1 -24265.332,E2 -24265.332} C_VEL
LIN {X 0,Y 206.654,Z 326.944,A -85,B 0,C 180,E1 -24266.057,E2 -24266.057} C_VEL
LIN {X 0,Y 208.785,Z 305.056,A -85,B 0,C 180,E1 -24266.687,E2 -24266.687} C_VEL
LIN {X 0,Y 212.362,Z 261.059,A -85,B 0,C 180,E1 -24267.888,E2 -24267.888} C_VEL
LIN {X 0,Y 208.256,Z 250.562,A -85,B 0,C 180,E1 -24270.426,E2 -24270.426} C_VEL
LIN {X 0,Y 204.234,Z 241.316,A -85,B 0,C 180,E1 -24273.152,E2 -24273.152} C_VEL
LIN {X 0,Y 200.866,Z 234.473,A -85,B 0,C 180,E1 -24275.667,E2 -24275.667} C_VEL
LIN {X 0,Y 196.894,Z 228.202,A -85,B 0,C 180,E1 -24278.944,E2 -24278.944} C_VEL
LIN {X 0,Y 194.448,Z 224.474,A -85,B 0,C 180,E1 -24281.291,E2 -24281.291} C_VEL
LIN {X 0,Y 191.876,Z 220.644,A -85,B 0,C 180,E1 -24284.176,E2 -24284.176} C_VEL
LIN {X 0,Y 189.459,Z 217.043,A -85,B 0,C 180,E1 -24287.549,E2 -24287.549} C_VEL
LIN {X 0,Y 188.911,Z 216.188,A -85,B 0,C 180,E1 -24288.465,E2 -24288.465} C_VEL
LIN {X 0,Y 186.776,Z 213.457,A -85,B 0,C 180,E1 -24292.976,E2 -24292.976} C_VEL
LIN {X 0,Y 186.141,Z 211.265,A -85,B 0,C 180,E1 -24295.67,E2 -24295.67} C_VEL
LIN {X 0,Y 185.605,Z 210.863,A -85,B 0,C 180,E1 -24300,E2 -24300} C_VEL
LIN {X 0,Y 186.174,Z 211.515,A -85,B 0,C 180,E1 -24305.008,E2 -24305.008} C_VEL
LIN {X 0,Y 187.661,Z 214.991,A -85,B 0,C 180,E1 -24309.702,E2 -24309.702} C_VEL
LIN {X 0,Y 189.237,Z 216.641,A -85,B 0,C 180,E1 -24312.517,E2 -24312.517} C_VEL
LIN {X 0,Y 191.414,Z 220.179,A -85,B 0,C 180,E1 -24315.711,E2 -24315.711} C_VEL
LIN {X 0,Y 192.475,Z 221.528,A -85,B 0,C 180,E1 -24316.985,E2 -24316.985} C_VEL
LIN {X 0,Y 195.541,Z 226.158,A -85,B 0,C 180,E1 -24320.239,E2 -24320.239} C_VEL
LIN {X 0,Y 198.245,Z 230.353,A -85,B 0,C 180,E1 -24322.677,E2 -24322.677} C_VEL
LIN {X 0,Y 202.188,Z 236.641,A -85,B 0,C 180,E1 -24325.755,E2 -24325.755} C_VEL
LIN {X 0,Y 206.535,Z 244.354,A -85,B 0,C 180,E1 -24328.728,E2 -24328.728} C_VEL
LIN {X 0,Y 211.465,Z 253.78,A -85,B 0,C 180,E1 -24331.704,E2 -24331.704} C_VEL
LIN {X 0,Y 212.667,Z 256.325,A -85,B 0,C 180,E1 -24332.387,E2 -24332.387} C_VEL
LIN {X 0,Y 207.489,Z 318.174,A -85,B 0,C 180,E1 -24334.113,E2 -24334.113} C_VEL
LIN {X 0,Y 205.077,Z 333.481,A -85,B 0,C 180,E1 -24334.773,E2 -24334.773} C_VEL
LIN {X 0,Y 201.826,Z 348.187,A -85,B 0,C 180,E1 -24335.729,E2 -24335.729} C_VEL
LIN {X 0,Y 197.682,Z 362.766,A -85,B 0,C 180,E1 -24337.046,E2 -24337.046} C_VEL
LIN {X 0,Y 193.219,Z 375.702,A -85,B 0,C 180,E1 -24338.603,E2 -24338.603} C_VEL
LIN {X 0,Y 187.441,Z 389.265,A -85,B 0,C 180,E1 -24340.601,E2 -24340.601} C_VEL
LIN {X 0,Y 181.857,Z 400.605,A -85,B 0,C 180,E1 -24342.754,E2 -24342.754} C_VEL
LIN {X 0,Y 175.497,Z 412.055,A -85,B 0,C 180,E1 -24345.508,E2 -24345.508} C_VEL
LIN {X 0,Y 169.557,Z 421.686,A -85,B 0,C 180,E1 -24348.456,E2 -24348.456} C_VEL
LIN {X 0,Y 164.217,Z 429.897,A -85,B 0,C 180,E1 -24351.643,E2 -24351.643} C_VEL
LIN {X 0,Y 158.461,Z 437.972,A -85,B 0,C 180,E1 -24355.564,E2 -24355.564} C_VEL
LIN {X 0,Y 153.435,Z 444.633,A -85,B 0,C 180,E1 -24359.745,E2 -24359.745} C_VEL
LIN {X 0,Y 148.735,Z 450.789,A -85,B 0,C 180,E1 -24364.833,E2 -24364.833} C_VEL
LIN {X 0,Y 145.115,Z 455.536,A -85,B 0,C 180,E1 -24370.183,E2 -24370.183} C_VEL
LIN {X 0,Y 142.705,Z 459.002,A -85,B 0,C 180,E1 -24375.745,E2 -24375.745} C_VEL
LIN {X 0,Y 141.255,Z 461.288,A -85,B 0,C 180,E1 -24381.416,E2 -24381.416} C_VEL
LIN {X 0,Y 140.677,Z 462.448,A -85,B 0,C 180,E1 -24387.137,E2 -24387.137} C_VEL
LIN {X 0,Y 140.653,Z 462.501,A -85,B 0,C 180,E1 -24392.077,E2 -24392.077} C_VEL
LIN {X 0,Y 140.866,Z 462.04,A -85,B 0,C 180,E1 -24395.727,E2 -24395.727} C_VEL
LIN {X 0,Y 141.841,Z 460.366,A -85,B 0,C 180,E1 -24401.432,E2 -24401.432} C_VEL
LIN {X 0,Y 143.735,Z 457.539,A -85,B 0,C 180,E1 -24407.06,E2 -24407.06} C_VEL
LIN {X 0,Y 146.813,Z 453.483,A -85,B 0,C 180,E1 -24412.518,E2 -24412.518} C_VEL
LIN {X 0,Y 150.863,Z 448.103,A -85,B 0,C 180,E1 -24417.766,E2 -24417.766} C_VEL
LIN {X 0,Y 156.136,Z 441.236,A -85,B 0,C 180,E1 -24422.694,E2 -24422.694} C_VEL
LIN {X 0,Y 162.381,Z 432.66,A -85,B 0,C 180,E1 -24427.296,E2 -24427.296} C_VEL
LIN {X 0,Y 168.656,Z 423.533,A -85,B 0,C 180,E1 -24431.02,E2 -24431.02} C_VEL
LIN {X 0,Y 174.353,Z 414.243,A -85,B 0,C 180,E1 -24434.054,E2 -24434.054} C_VEL
LIN {X 0,Y 181.205,Z 402.2,A -85,B 0,C 180,E1 -24437.06,E2 -24437.06} C_VEL
LIN {X 0,Y 187.34,Z 389.897,A -85,B 0,C 180,E1 -24439.436,E2 -24439.436} C_VEL
LIN {X 0,Y 193.039,Z 376.51,A -85,B 0,C 180,E1 -24441.461,E2 -24441.461} C_VEL
LIN {X 0,Y 197.194,Z 364.733,A -85,B 0,C 180,E1 -24442.887,E2 -24442.887} C_VEL
LIN {X 0,Y 201.452,Z 350.454,A -85,B 0,C 180,E1 -24444.206,E2 -24444.206} C_VEL
LIN {X 0,Y 204.835,Z 335.746,A -85,B 0,C 180,E1 -24445.217,E2 -24445.217} C_VEL
LIN {X 0,Y 207.442,Z 320.162,A -85,B 0,C 180,E1 -24445.932,E2 -24445.932} C_VEL
LIN {X 0,Y 209.697,Z 295.481,A -85,B 0,C 180,E1 -24446.671,E2 -24446.671} C_VEL
LIN {X 0,Y 212.903,Z 256.547,A -85,B 0,C 180,E1 -24447.718,E2 -24447.718} C_VEL
LIN {X 0,Y 208.102,Z 247.04,A -85,B 0,C 180,E1 -24450.541,E2 -24450.541} C_VEL
LIN {X 0,Y 203.644,Z 238.965,A -85,B 0,C 180,E1 -24453.483,E2 -24453.483} C_VEL
LIN {X 0,Y 199.598,Z 232.255,A -85,B 0,C 180,E1 -24456.526,E2 -24456.526} C_VEL
LIN {X 0,Y 196.512,Z 227.588,A -85,B 0,C 180,E1 -24459.182,E2 -24459.182} C_VEL
LIN {X 0,Y 194.746,Z 224.859,A -85,B 0,C 180,E1 -24460.91,E2 -24460.91} C_VEL
LIN {X 0,Y 192.066,Z 220.803,A -85,B 0,C 180,E1 -24463.935,E2 -24463.935} C_VEL
LIN {X 0,Y 189.629,Z 217.312,A -85,B 0,C 180,E1 -24467.356,E2 -24467.356} C_VEL
LIN {X 0,Y 188.992,Z 216.202,A -85,B 0,C 180,E1 -24468.47,E2 -24468.47} C_VEL
LIN {X 0,Y 186.945,Z 213.587,A -85,B 0,C 180,E1 -24472.982,E2 -24472.982} C_VEL
LIN {X 0,Y 186.263,Z 211.306,A -85,B 0,C 180,E1 -24476.214,E2 -24476.214} C_VEL
LIN {X 0,Y 185.938,Z 210.947,A -85,B 0,C 180,E1 -24480,E2 -24480} C_VEL
LIN {X 0,Y 186.322,Z 211.435,A -85,B 0,C 180,E1 -24483.785,E2 -24483.785} C_VEL
LIN {X 0,Y 188.036,Z 215.333,A -85,B 0,C 180,E1 -24489.433,E2 -24489.433} C_VEL
LIN {X 0,Y 189.347,Z 216.613,A -85,B 0,C 180,E1 -24491.779,E2 -24491.779} C_VEL
LIN {X 0,Y 191.813,Z 220.486,A -85,B 0,C 180,E1 -24495.405,E2 -24495.405} C_VEL
LIN {X 0,Y 193.071,Z 222.395,A -85,B 0,C 180,E1 -24496.93,E2 -24496.93} C_VEL
LIN {X 0,Y 195.723,Z 226.247,A -85,B 0,C 180,E1 -24499.706,E2 -24499.706} C_VEL
LIN {X 0,Y 198.722,Z 230.969,A -85,B 0,C 180,E1 -24502.413,E2 -24502.413} C_VEL
LIN {X 0,Y 201.708,Z 235.807,A -85,B 0,C 180,E1 -24504.775,E2 -24504.775} C_VEL
LIN {X 0,Y 205.511,Z 243.87,A -85,B 0,C 180,E1 -24507.564,E2 -24507.564} C_VEL
LIN {X 0,Y 210.01,Z 254.535,A -85,B 0,C 180,E1 -24510.521,E2 -24510.521} C_VEL
LIN {X 0,Y 212.561,Z 261.226,A -85,B 0,C 180,E1 -24512.078,E2 -24512.078} C_VEL
LIN {X 0,Y 207.22,Z 324.847,A -85,B 0,C 180,E1 -24513.85,E2 -24513.85} C_VEL
LIN {X 0,Y 204.678,Z 340.424,A -85,B 0,C 180,E1 -24514.504,E2 -24514.504} C_VEL
LIN {X 0,Y 201.125,Z 355.653,A -85,B 0,C 180,E1 -24515.45,E2 -24515.45} C_VEL
LIN {X 0,Y 196.925,Z 369.376,A -85,B 0,C 180,E1 -24516.582,E2 -24516.582} C_VEL
LIN {X 0,Y 192.012,Z 382.827,A -85,B 0,C 180,E1 -24518.099,E2 -24518.099} C_VEL
LIN {X 0,Y 186.74,Z 395.113,A -85,B 0,C 180,E1 -24519.89,E2 -24519.89} C_VEL
LIN {X 0,Y 182.277,Z 404.329,A -85,B 0,C 180,E1 -24521.54,E2 -24521.54} C_VEL
LIN {X 0,Y 179.39,Z 408.923,A -85,B 0,C 180,E1 -24522.313,E2 -24522.313} C_VEL
LIN {X 0,Y 168.199,Z 421.594,A -85,B 0,C 180,E1 -24524.207,E2 -24524.207} C_VEL
LIN {X 0,Y 164.894,Z 425.568,A -85,B 0,C 180,E1 -24525.179,E2 -24525.179} C_VEL
LIN {X 0,Y 163.984,Z 426.851,A -85,B 0,C 180,E1 -24525.587,E2 -24525.587} C_VEL
LIN {X 0,Y 157.95,Z 435.682,A -85,B 0,C 180,E1 -24528.887,E2 -24528.887} C_VEL
LIN {X 0,Y 151.853,Z 444.16,A -85,B 0,C 180,E1 -24533.011,E2 -24533.011} C_VEL
LIN {X 0,Y 145.66,Z 451.981,A -85,B 0,C 180,E1 -24537.944,E2 -24537.944} C_VEL
LIN {X 0,Y 140.8,Z 458.216,A -85,B 0,C 180,E1 -24543.305,E2 -24543.305} C_VEL
LIN {X 0,Y 137.155,Z 463.046,A -85,B 0,C 180,E1 -24548.98,E2 -24548.98} C_VEL
LIN {X 0,Y 134.714,Z 466.592,A -85,B 0,C 180,E1 -24554.879,E2 -24554.879} C_VEL
LIN {X 0,Y 133.568,Z 468.935,A -85,B 0,C 180,E1 -24560.918,E2 -24560.918} C_VEL
LIN {X 0,Y 133.389,Z 470.12,A -85,B 0,C 180,E1 -24566.98,E2 -24566.98} C_VEL
LIN {X 0,Y 133.531,Z 470.279,A -85,B 0,C 180,E1 -24570,E2 -24570} C_VEL
LIN {X 0,Y 133.374,Z 469.652,A -85,B 0,C 180,E1 -24576.049,E2 -24576.049} C_VEL
LIN {X 0,Y 133.993,Z 467.867,A -85,B 0,C 180,E1 -24582.111,E2 -24582.111} C_VEL
LIN {X 0,Y 135.774,Z 464.911,A -85,B 0,C 180,E1 -24588.094,E2 -24588.094} C_VEL
LIN {X 0,Y 138.748,Z 460.714,A -85,B 0,C 180,E1 -24593.905,E2 -24593.905} C_VEL
LIN {X 0,Y 143.042,Z 455.172,A -85,B 0,C 180,E1 -24599.428,E2 -24599.428} C_VEL
LIN {X 0,Y 148.551,Z 448.135,A -85,B 0,C 180,E1 -24604.592,E2 -24604.592} C_VEL
LIN {X 0,Y 154.222,Z 440.616,A -85,B 0,C 180,E1 -24608.8,E2 -24608.8} C_VEL
LIN {X 0,Y 160.628,Z 431.555,A -85,B 0,C 180,E1 -24612.701,E2 -24612.701} C_VEL
LIN {X 0,Y 167.845,Z 420.675,A -85,B 0,C 180,E1 -24616.244,E2 -24616.244} C_VEL
LIN {X 0,Y 173.381,Z 411.436,A -85,B 0,C 180,E1 -24618.582,E2 -24618.582} C_VEL
LIN {X 0,Y 179.822,Z 399.565,A -85,B 0,C 180,E1 -24620.966,E2 -24620.966} C_VEL
LIN {X 0,Y 185.832,Z 386.575,A -85,B 0,C 180,E1 -24623.028,E2 -24623.028} C_VEL
LIN {X 0,Y 190.832,Z 373.991,A -85,B 0,C 180,E1 -24624.57,E2 -24624.57} C_VEL
LIN {X 0,Y 195.719,Z 359.328,A -85,B 0,C 180,E1 -24625.908,E2 -24625.908} C_VEL
LIN {X 0,Y 199.728,Z 343.937,A -85,B 0,C 180,E1 -24626.921,E2 -24626.921} C_VEL
LIN {X 0,Y 202.516,Z 328.544,A -85,B 0,C 180,E1 -24627.653,E2 -24627.653} C_VEL
LIN {X 0,Y 204.476,Z 310.543,A -85,B 0,C 180,E1 -24628.198,E2 -24628.198} C_VEL
LIN {X 0,Y 208.447,Z 263.989,A -85,B 0,C 180,E1 -24629.437,E2 -24629.437} C_VEL
LIN {X 0,Y 205.013,Z 254.915,A -85,B 0,C 180,E1 -24631.735,E2 -24631.735} C_VEL
LIN {X 0,Y 201.375,Z 246.223,A -85,B 0,C 180,E1 -24634.394,E2 -24634.394} C_VEL
LIN {X 0,Y 198.678,Z 240.506,A -85,B 0,C 180,E1 -24636.55,E2 -24636.55} C_VEL
LIN {X 0,Y 195.061,Z 234.548,A -85,B 0,C 180,E1 -24639.709,E2 -24639.709} C_VEL
LIN {X 0,Y 192.751,Z 230.917,A -85,B 0,C 180,E1 -24642.052,E2 -24642.052} C_VEL
LIN {X 0,Y 190.477,Z 227.343,A -85,B 0,C 180,E1 -24644.754,E2 -24644.754} C_VEL
LIN {X 0,Y 188.258,Z 223.896,A -85,B 0,C 180,E1 -24648.015,E2 -24648.015} C_VEL
LIN {X 0,Y 187.584,Z 222.887,A -85,B 0,C 180,E1 -24649.203,E2 -24649.203} C_VEL
LIN {X 0,Y 185.653,Z 220.09,A -85,B 0,C 180,E1 -24653.752,E2 -24653.752} C_VEL
LIN {X 0,Y 185.156,Z 218.237,A -85,B 0,C 180,E1 -24656.192,E2 -24656.192} C_VEL
LIN {X 0,Y 184.74,Z 217.908,A -85,B 0,C 180,E1 -24660,E2 -24660} C_VEL
LIN {X 0,Y 185.218,Z 218.466,A -85,B 0,C 180,E1 -24664.625,E2 -24664.625} C_VEL
LIN {X 0,Y 186.67,Z 221.998,A -85,B 0,C 180,E1 -24669.481,E2 -24669.481} C_VEL
LIN {X 0,Y 188.016,Z 223.472,A -85,B 0,C 180,E1 -24672,E2 -24672} C_VEL
LIN {X 0,Y 190.143,Z 227.007,A -85,B 0,C 180,E1 -24675.269,E2 -24675.269} C_VEL
LIN {X 0,Y 191.156,Z 228.497,A -85,B 0,C 180,E1 -24676.555,E2 -24676.555} C_VEL
LIN {X 0,Y 193.847,Z 232.63,A -85,B 0,C 180,E1 -24679.539,E2 -24679.539} C_VEL
LIN {X 0,Y 196.711,Z 237.295,A -85,B 0,C 180,E1 -24682.242,E2 -24682.242} C_VEL
LIN {X 0,Y 200.2,Z 243.118,A -85,B 0,C 180,E1 -24685.083,E2 -24685.083} C_VEL
LIN {X 0,Y 204.642,Z 251.287,A -85,B 0,C 180,E1 -24688.248,E2 -24688.248} C_VEL
LIN {X 0,Y 208.758,Z 259.657,A -85,B 0,C 180,E1 -24690.859,E2 -24690.859} C_VEL
LIN {X 0,Y 203.551,Z 318.786,A -85,B 0,C 180,E1 -24692.481,E2 -24692.481} C_VEL
LIN {X 0,Y 200.952,Z 334.46,A -85,B 0,C 180,E1 -24693.156,E2 -24693.156} C_VEL
LIN {X 0,Y 197.763,Z 348.394,A -85,B 0,C 180,E1 -24694.058,E2 -24694.058} C_VEL
LIN {X 0,Y 193.49,Z 362.97,A -85,B 0,C 180,E1 -24695.37,E2 -24695.37} C_VEL
LIN {X 0,Y 188.743,Z 376.237,A -85,B 0,C 180,E1 -24696.961,E2 -24696.961} C_VEL
LIN {X 0,Y 182.906,Z 389.468,A -85,B 0,C 180,E1 -24698.914,E2 -24698.914} C_VEL
LIN {X 0,Y 177.098,Z 400.808,A -85,B 0,C 180,E1 -24701.062,E2 -24701.062} C_VEL
LIN {X 0,Y 170.503,Z 412.256,A -85,B 0,C 180,E1 -24703.835,E2 -24703.835} C_VEL
LIN {X 0,Y 164.279,Z 421.889,A -85,B 0,C 180,E1 -24706.804,E2 -24706.804} C_VEL
LIN {X 0,Y 158.709,Z 430.098,A -85,B 0,C 180,E1 -24710.052,E2 -24710.052} C_VEL
LIN {X 0,Y 152.64,Z 438.173,A -85,B 0,C 180,E1 -24714.052,E2 -24714.052} C_VEL
LIN {X 0,Y 147.309,Z 444.834,A -85,B 0,C 180,E1 -24718.345,E2 -24718.345} C_VEL
LIN {X 0,Y 142.299,Z 450.99,A -85,B 0,C 180,E1 -24723.609,E2 -24723.609} C_VEL
LIN {X 0,Y 138.431,Z 455.736,A -85,B 0,C 180,E1 -24729.183,E2 -24729.183} C_VEL
LIN {X 0,Y 135.808,Z 459.203,A -85,B 0,C 180,E1 -24735.004,E2 -24735.004} C_VEL
LIN {X 0,Y 134.217,Z 461.488,A -85,B 0,C 180,E1 -24740.962,E2 -24740.962} C_VEL
LIN {X 0,Y 133.602,Z 462.646,A -85,B 0,C 180,E1 -24746.985,E2 -24746.985} C_VEL
LIN {X 0,Y 133.56,Z 462.751,A -85,B 0,C 180,E1 -24751.167,E2 -24751.167} C_VEL
LIN {X 0,Y 133.807,Z 462.238,A -85,B 0,C 180,E1 -24756.03,E2 -24756.03} C_VEL
LIN {X 0,Y 134.877,Z 460.565,A -85,B 0,C 180,E1 -24762.03,E2 -24762.03} C_VEL
LIN {X 0,Y 136.917,Z 457.739,A -85,B 0,C 180,E1 -24767.938,E2 -24767.938} C_VEL
LIN {X 0,Y 140.25,Z 453.682,A -85,B 0,C 180,E1 -24773.634,E2 -24773.634} C_VEL
LIN {X 0,Y 144.583,Z 448.302,A -85,B 0,C 180,E1 -24779.084,E2 -24779.084} C_VEL
LIN {X 0,Y 150.185,Z 441.434,A -85,B 0,C 180,E1 -24784.163,E2 -24784.163} C_VEL
LIN {X 0,Y 156.771,Z 432.857,A -85,B 0,C 180,E1 -24788.875,E2 -24788.875} C_VEL
LIN {X 0,Y 162.387,Z 425.141,A -85,B 0,C 180,E1 -24792.132,E2 -24792.132} C_VEL
LIN {X 0,Y 168.26,Z 416.059,A -85,B 0,C 180,E1 -24795.241,E2 -24795.241} C_VEL
LIN {X 0,Y 174.792,Z 405.331,A -85,B 0,C 180,E1 -24798.06,E2 -24798.06} C_VEL
LIN {X 0,Y 181,Z 393.619,A -85,B 0,C 180,E1 -24800.509,E2 -24800.509} C_VEL
LIN {X 0,Y 187.273,Z 380.13,A -85,B 0,C 180,E1 -24802.661,E2 -24802.661} C_VEL
LIN {X 0,Y 192.365,Z 366.688,A -85,B 0,C 180,E1 -24804.381,E2 -24804.381} C_VEL
LIN {X 0,Y 196.742,Z 352.901,A -85,B 0,C 180,E1 -24805.698,E2 -24805.698} C_VEL
LIN {X 0,Y 200.558,Z 337.456,A -85,B 0,C 180,E1 -24806.787,E2 -24806.787} C_VEL
LIN {X 0,Y 203.394,Z 321.471,A -85,B 0,C 180,E1 -24807.543,E2 -24807.543} C_VEL
LIN {X 0,Y 205.512,Z 300.34,A -85,B 0,C 180,E1 -24808.184,E2 -24808.184} C_VEL
LIN {X 0,Y 208.984,Z 260.034,A -85,B 0,C 180,E1 -24809.241,E2 -24809.241} C_VEL
LIN {X 0,Y 205.08,Z 251.915,A -85,B 0,C 180,E1 -24811.726,E2 -24811.726} C_VEL
LIN {X 0,Y 200.805,Z 243.992,A -85,B 0,C 180,E1 -24814.751,E2 -24814.751} C_VEL
LIN {X 0,Y 197.076,Z 237.705,A -85,B 0,C 180,E1 -24817.769,E2 -24817.769} C_VEL
LIN {X 0,Y 194.467,Z 233.537,A -85,B 0,C 180,E1 -24820.194,E2 -24820.194} C_VEL
LIN {X 0,Y 192.906,Z 231.108,A -85,B 0,C 180,E1 -24821.823,E2 -24821.823} C_VEL
LIN {X 0,Y 190.636,Z 227.487,A -85,B 0,C 180,E1 -24824.556,E2 -24824.556} C_VEL
LIN {X 0,Y 188.255,Z 223.783,A -85,B 0,C 180,E1 -24828.151,E2 -24828.151} C_VEL
LIN {X 0,Y 187.825,Z 223.074,A -85,B 0,C 180,E1 -24828.944,E2 -24828.944} C_VEL
LIN {X 0,Y 185.838,Z 220.26,A -85,B 0,C 180,E1 -24833.748,E2 -24833.748} C_VEL
LIN {X 0,Y 185.393,Z 218.409,A -85,B 0,C 180,E1 -24836.196,E2 -24836.196} C_VEL
LIN {X 0,Y 185.072,Z 217.995,A -85,B 0,C 180,E1 -24840,E2 -24840} C_VEL
LIN {X 0,Y 185.398,Z 218.492,A -85,B 0,C 180,E1 -24843.531,E2 -24843.531} C_VEL
LIN {X 0,Y 187.173,Z 222.462,A -85,B 0,C 180,E1 -24849.477,E2 -24849.477} C_VEL
LIN {X 0,Y 188.245,Z 223.68,A -85,B 0,C 180,E1 -24851.466,E2 -24851.466} C_VEL
LIN {X 0,Y 190.743,Z 227.54,A -85,B 0,C 180,E1 -24855.22,E2 -24855.22} C_VEL
LIN {X 0,Y 194.048,Z 232.782,A -85,B 0,C 180,E1 -24859.024,E2 -24859.024} C_VEL
LIN {X 0,Y 196.622,Z 236.974,A -85,B 0,C 180,E1 -24861.483,E2 -24861.483} C_VEL
LIN {X 0,Y 199.449,Z 241.709,A -85,B 0,C 180,E1 -24863.857,E2 -24863.857} C_VEL
LIN {X 0,Y 203.203,Z 250.122,A -85,B 0,C 180,E1 -24866.781,E2 -24866.781} C_VEL
LIN {X 0,Y 207.401,Z 260.71,A -85,B 0,C 180,E1 -24869.708,E2 -24869.708} C_VEL
LIN {X 0,Y 208.651,Z 264.079,A -85,B 0,C 180,E1 -24870.523,E2 -24870.523} C_VEL
LIN {X 0,Y 203.304,Z 324.95,A -85,B 0,C 180,E1 -24872.197,E2 -24872.197} C_VEL
LIN {X 0,Y 200.742,Z 340.234,A -85,B 0,C 180,E1 -24872.834,E2 -24872.834} C_VEL
LIN {X 0,Y 197.089,Z 355.461,A -85,B 0,C 180,E1 -24873.767,E2 -24873.767} C_VEL
LIN {X 0,Y 192.771,Z 369.183,A -85,B 0,C 180,E1 -24874.884,E2 -24874.884} C_VEL
LIN {X 0,Y 187.7,Z 382.633,A -85,B 0,C 180,E1 -24876.388,E2 -24876.388} C_VEL
LIN {X 0,Y 181.845,Z 395.795,A -85,B 0,C 180,E1 -24878.311,E2 -24878.311} C_VEL
LIN {X 0,Y 175.111,Z 408.745,A -85,B 0,C 180,E1 -24880.752,E2 -24880.752} C_VEL
LIN {X 0,Y 168.932,Z 419.152,A -85,B 0,C 180,E1 -24883.277,E2 -24883.277} C_VEL
LIN {X 0,Y 163.984,Z 426.851,A -85,B 0,C 180,E1 -24885.587,E2 -24885.587} C_VEL
LIN {X 0,Y 160.956,Z 430.688,A -85,B 0,C 180,E1 -24886.776,E2 -24886.776} C_VEL
LIN {X 0,Y 154.632,Z 436.621,A -85,B 0,C 180,E1 -24888.499,E2 -24888.499} C_VEL
LIN {X 0,Y 148.24,Z 442.14,A -85,B 0,C 180,E1 -24890.461,E2 -24890.461} C_VEL
LIN {X 0,Y 145.18,Z 445.205,A -85,B 0,C 180,E1 -24892.03,E2 -24892.03} C_VEL
LIN {X 0,Y 139.64,Z 451.782,A -85,B 0,C 180,E1 -24896.384,E2 -24896.384} C_VEL
LIN {X 0,Y 134.425,Z 458.016,A -85,B 0,C 180,E1 -24901.93,E2 -24901.93} C_VEL
LIN {X 0,Y 130.495,Z 462.846,A -85,B 0,C 180,E1 -24907.852,E2 -24907.852} C_VEL
LIN {X 0,Y 127.81,Z 466.392,A -85,B 0,C 180,E1 -24914.041,E2 -24914.041} C_VEL
LIN {X 0,Y 126.529,Z 468.736,A -85,B 0,C 180,E1 -24920.408,E2 -24920.408} C_VEL
LIN {X 0,Y 126.293,Z 469.921,A -85,B 0,C 180,E1 -24926.81,E2 -24926.81} C_VEL
LIN {X 0,Y 126.427,Z 470.08,A -85,B 0,C 180,E1 -24930,E2 -24930} C_VEL
LIN {X 0,Y 126.293,Z 469.915,A -85,B 0,C 180,E1 -24933.19,E2 -24933.19} C_VEL
LIN {X 0,Y 126.527,Z 468.704,A -85,B 0,C 180,E1 -24939.592,E2 -24939.592} C_VEL
LIN {X 0,Y 127.786,Z 466.336,A -85,B 0,C 180,E1 -24945.961,E2 -24945.961} C_VEL
LIN {X 0,Y 130.445,Z 462.772,A -85,B 0,C 180,E1 -24952.157,E2 -24952.157} C_VEL
LIN {X 0,Y 134.387,Z 457.918,A -85,B 0,C 180,E1 -24958.078,E2 -24958.078} C_VEL
LIN {X 0,Y 139.588,Z 451.648,A -85,B 0,C 180,E1 -24963.63,E2 -24963.63} C_VEL
LIN {X 0,Y 146.13,Z 443.793,A -85,B 0,C 180,E1 -24968.699,E2 -24968.699} C_VEL
LIN {X 0,Y 152.454,Z 435.438,A -85,B 0,C 180,E1 -24972.84,E2 -24972.84} C_VEL
LIN {X 0,Y 159.662,Z 425.383,A -85,B 0,C 180,E1 -24976.577,E2 -24976.577} C_VEL
LIN {X 0,Y 166.353,Z 415.114,A -85,B 0,C 180,E1 -24979.504,E2 -24979.504} C_VEL
LIN {X 0,Y 173.579,Z 402.875,A -85,B 0,C 180,E1 -24982.142,E2 -24982.142} C_VEL
LIN {X 0,Y 179.973,Z 390.048,A -85,B 0,C 180,E1 -24984.322,E2 -24984.322} C_VEL
LIN {X 0,Y 186.155,Z 375.556,A -85,B 0,C 180,E1 -24986.158,E2 -24986.158} C_VEL
LIN {X 0,Y 191.161,Z 361.382,A -85,B 0,C 180,E1 -24987.49,E2 -24987.49} C_VEL
LIN {X 0,Y 195.433,Z 346.018,A -85,B 0,C 180,E1 -24988.535,E2 -24988.535} C_VEL
LIN {X 0,Y 198.448,Z 330.824,A -85,B 0,C 180,E1 -24989.286,E2 -24989.286} C_VEL
LIN {X 0,Y 200.466,Z 314.644,A -85,B 0,C 180,E1 -24989.795,E2 -24989.795} C_VEL
LIN {X 0,Y 204.657,Z 266.787,A -85,B 0,C 180,E1 -24991.069,E2 -24991.069} C_VEL
LIN {X 0,Y 200.798,Z 256.44,A -85,B 0,C 180,E1 -24993.916,E2 -24993.916} C_VEL
LIN {X 0,Y 197.364,Z 248.209,A -85,B 0,C 180,E1 -24996.737,E2 -24996.737} C_VEL
LIN {X 0,Y 195.219,Z 244.172,A -85,B 0,C 180,E1 -24998.623,E2 -24998.623} C_VEL
LIN {X 0,Y 191.786,Z 238.268,A -85,B 0,C 180,E1 -25002.065,E2 -25002.065} C_VEL
LIN {X 0,Y 189.004,Z 233.933,A -85,B 0,C 180,E1 -25005.464,E2 -25005.464} C_VEL
LIN {X 0,Y 186.573,Z 229.889,A -85,B 0,C 180,E1 -25009.419,E2 -25009.419} C_VEL
LIN {X 0,Y 184.628,Z 226.924,A -85,B 0,C 180,E1 -25014.266,E2 -25014.266} C_VEL
LIN {X 0,Y 184.184,Z 225.226,A -85,B 0,C 180,E1 -25016.719,E2 -25016.719} C_VEL
LIN {X 0,Y 183.875,Z 224.957,A -85,B 0,C 180,E1 -25020,E2 -25020} C_VEL
LIN {X 0,Y 184.286,Z 225.541,A -85,B 0,C 180,E1 -25024.375,E2 -25024.375} C_VEL
LIN {X 0,Y 185.683,Z 228.995,A -85,B 0,C 180,E1 -25029.257,E2 -25029.257} C_VEL
LIN {X 0,Y 186.883,Z 230.425,A -85,B 0,C 180,E1 -25031.61,E2 -25031.61} C_VEL
LIN {X 0,Y 189.08,Z 234.07,A -85,B 0,C 180,E1 -25035.081,E2 -25035.081} C_VEL
LIN {X 0,Y 192.254,Z 239.222,A -85,B 0,C 180,E1 -25038.904,E2 -25038.904} C_VEL
LIN {X 0,Y 195.937,Z 245.403,A -85,B 0,C 180,E1 -25042.458,E2 -25042.458} C_VEL
LIN {X 0,Y 200.216,Z 253.287,A -85,B 0,C 180,E1 -25045.93,E2 -25045.93} C_VEL
LIN {X 0,Y 204.629,Z 262.353,A -85,B 0,C 180,E1 -25049.041,E2 -25049.041} C_VEL
LIN {X 0,Y 204.937,Z 262.995,A -85,B 0,C 180,E1 -25049.242,E2 -25049.242} C_VEL
LIN {X 0,Y 199.859,Z 318.798,A -85,B 0,C 180,E1 -25050.756,E2 -25050.756} C_VEL
LIN {X 0,Y 197.169,Z 334.668,A -85,B 0,C 180,E1 -25051.434,E2 -25051.434} C_VEL
LIN {X 0,Y 193.562,Z 349.753,A -85,B 0,C 180,E1 -25052.416,E2 -25052.416} C_VEL
LIN {X 0,Y 189.475,Z 363.175,A -85,B 0,C 180,E1 -25053.621,E2 -25053.621} C_VEL
LIN {X 0,Y 184.454,Z 376.702,A -85,B 0,C 180,E1 -25055.231,E2 -25055.231} C_VEL
LIN {X 0,Y 178.534,Z 389.671,A -85,B 0,C 180,E1 -25057.142,E2 -25057.142} C_VEL
LIN {X 0,Y 172.506,Z 401.011,A -85,B 0,C 180,E1 -25059.279,E2 -25059.279} C_VEL
LIN {X 0,Y 165.652,Z 412.459,A -85,B 0,C 180,E1 -25062.059,E2 -25062.059} C_VEL
LIN {X 0,Y 159.152,Z 422.091,A -85,B 0,C 180,E1 -25065.045,E2 -25065.045} C_VEL
LIN {X 0,Y 153.334,Z 430.299,A -85,B 0,C 180,E1 -25068.348,E2 -25068.348} C_VEL
LIN {X 0,Y 146.923,Z 438.375,A -85,B 0,C 180,E1 -25072.418,E2 -25072.418} C_VEL
LIN {X 0,Y 141.289,Z 445.035,A -85,B 0,C 180,E1 -25076.827,E2 -25076.827} C_VEL
LIN {X 0,Y 135.938,Z 451.192,A -85,B 0,C 180,E1 -25082.27,E2 -25082.27} C_VEL
LIN {X 0,Y 131.8,Z 455.937,A -85,B 0,C 180,E1 -25088.083,E2 -25088.083} C_VEL
LIN {X 0,Y 128.945,Z 459.403,A -85,B 0,C 180,E1 -25094.186,E2 -25094.186} C_VEL
LIN {X 0,Y 127.194,Z 461.687,A -85,B 0,C 180,E1 -25100.459,E2 -25100.459} C_VEL
LIN {X 0,Y 126.513,Z 462.845,A -85,B 0,C 180,E1 -25106.816,E2 -25106.816} C_VEL
LIN {X 0,Y 126.505,Z 462.997,A -85,B 0,C 180,E1 -25110,E2 -25110} C_VEL
LIN {X 0,Y 126.743,Z 462.437,A -85,B 0,C 180,E1 -25116.367,E2 -25116.367} C_VEL
LIN {X 0,Y 127.915,Z 460.764,A -85,B 0,C 180,E1 -25122.696,E2 -25122.696} C_VEL
LIN {X 0,Y 130.138,Z 457.938,A -85,B 0,C 180,E1 -25128.907,E2 -25128.907} C_VEL
LIN {X 0,Y 133.749,Z 453.88,A -85,B 0,C 180,E1 -25134.858,E2 -25134.858} C_VEL
LIN {X 0,Y 138.393,Z 448.5,A -85,B 0,C 180,E1 -25140.52,E2 -25140.52} C_VEL
LIN {X 0,Y 144.342,Z 441.632,A -85,B 0,C 180,E1 -25145.752,E2 -25145.752} C_VEL
LIN {X 0,Y 151.289,Z 433.055,A -85,B 0,C 180,E1 -25150.569,E2 -25150.569} C_VEL
LIN {X 0,Y 157.828,Z 424.408,A -85,B 0,C 180,E1 -25154.244,E2 -25154.244} C_VEL
LIN {X 0,Y 164.426,Z 414.636,A -85,B 0,C 180,E1 -25157.503,E2 -25157.503} C_VEL
LIN {X 0,Y 171.828,Z 402.591,A -85,B 0,C 180,E1 -25160.535,E2 -25160.535} C_VEL
LIN {X 0,Y 178.432,Z 390.286,A -85,B 0,C 180,E1 -25162.902,E2 -25162.902} C_VEL
LIN {X 0,Y 184.56,Z 376.819,A -85,B 0,C 180,E1 -25164.921,E2 -25164.921} C_VEL
LIN {X 0,Y 189.622,Z 363.346,A -85,B 0,C 180,E1 -25166.505,E2 -25166.505} C_VEL
LIN {X 0,Y 194.157,Z 348.551,A -85,B 0,C 180,E1 -25167.792,E2 -25167.792} C_VEL
LIN {X 0,Y 197.776,Z 332.892,A -85,B 0,C 180,E1 -25168.776,E2 -25168.776} C_VEL
LIN {X 0,Y 200.21,Z 317.988,A -85,B 0,C 180,E1 -25169.392,E2 -25169.392} C_VEL
LIN {X 0,Y 205.164,Z 263.182,A -85,B 0,C 180,E1 -25170.874,E2 -25170.874} C_VEL
LIN {X 0,Y 201.199,Z 255.044,A -85,B 0,C 180,E1 -25173.623,E2 -25173.623} C_VEL
LIN {X 0,Y 197.48,Z 247.973,A -85,B 0,C 180,E1 -25176.537,E2 -25176.537} C_VEL
LIN {X 0,Y 193.831,Z 241.625,A -85,B 0,C 180,E1 -25179.85,E2 -25179.85} C_VEL
LIN {X 0,Y 191.23,Z 237.492,A -85,B 0,C 180,E1 -25182.626,E2 -25182.626} C_VEL
LIN {X 0,Y 189.217,Z 234.136,A -85,B 0,C 180,E1 -25185.205,E2 -25185.205} C_VEL
LIN {X 0,Y 186.82,Z 230.052,A -85,B 0,C 180,E1 -25189.158,E2 -25189.158} C_VEL
LIN {X 0,Y 184.962,Z 227.435,A -85,B 0,C 180,E1 -25193.718,E2 -25193.718} C_VEL
LIN {X 0,Y 184.439,Z 225.346,A -85,B 0,C 180,E1 -25196.723,E2 -25196.723} C_VEL
LIN {X 0,Y 184.207,Z 225.043,A -85,B 0,C 180,E1 -25200,E2 -25200} C_VEL
LIN {X 0,Y 184.484,Z 225.507,A -85,B 0,C 180,E1 -25203.276,E2 -25203.276} C_VEL
LIN {X 0,Y 186.169,Z 229.444,A -85,B 0,C 180,E1 -25209.232,E2 -25209.232} C_VEL
LIN {X 0,Y 186.995,Z 230.338,A -85,B 0,C 180,E1 -25210.831,E2 -25210.831} C_VEL
LIN {X 0,Y 189.844,Z 235.129,A -85,B 0,C 180,E1 -25215.293,E2 -25215.293} C_VEL
LIN {X 0,Y 192.479,Z 239.408,A -85,B 0,C 180,E1 -25218.41,E2 -25218.41} C_VEL
LIN {X 0,Y 194.982,Z 243.697,A -85,B 0,C 180,E1 -25220.92,E2 -25220.92} C_VEL
LIN {X 0,Y 197.393,Z 247.992,A -85,B 0,C 180,E1 -25223.057,E2 -25223.057} C_VEL
LIN {X 0,Y 200.871,Z 256.258,A -85,B 0,C 180,E1 -25225.934,E2 -25225.934} C_VEL
LIN {X 0,Y 204.557,Z 266.147,A -85,B 0,C 180,E1 -25228.68,E2 -25228.68} C_VEL
LIN {X 0,Y 204.895,Z 267.075,A -85,B 0,C 180,E1 -25228.917,E2 -25228.917} C_VEL
LIN {X 0,Y 199.672,Z 324.359,A -85,B 0,C 180,E1 -25230.458,E2 -25230.458} C_VEL
LIN {X 0,Y 196.986,Z 340.045,A -85,B 0,C 180,E1 -25231.1,E2 -25231.1} C_VEL
LIN {X 0,Y 193.232,Z 355.269,A -85,B 0,C 180,E1 -25232.016,E2 -25232.016} C_VEL
LIN {X 0,Y 188.806,Z 368.99,A -85,B 0,C 180,E1 -25233.12,E2 -25233.12} C_VEL
LIN {X 0,Y 183.564,Z 382.438,A -85,B 0,C 180,E1 -25234.598,E2 -25234.598} C_VEL
LIN {X 0,Y 177.07,Z 396.508,A -85,B 0,C 180,E1 -25236.653,E2 -25236.653} C_VEL
LIN {X 0,Y 169.951,Z 409.557,A -85,B 0,C 180,E1 -25239.161,E2 -25239.161} C_VEL
LIN {X 0,Y 163.007,Z 420.717,A -85,B 0,C 180,E1 -25241.949,E2 -25241.949} C_VEL
LIN {X 0,Y 156.503,Z 430.115,A -85,B 0,C 180,E1 -25244.986,E2 -25244.986} C_VEL
LIN {X 0,Y 149.696,Z 439.369,A -85,B 0,C 180,E1 -25248.907,E2 -25248.907} C_VEL
LIN {X 0,Y 145.18,Z 445.205,A -85,B 0,C 180,E1 -25252.03,E2 -25252.03} C_VEL
LIN {X 0,Y 142.153,Z 448.17,A -85,B 0,C 180,E1 -25253.699,E2 -25253.699} C_VEL
LIN {X 0,Y 135.872,Z 452.608,A -85,B 0,C 180,E1 -25256.287,E2 -25256.287} C_VEL
LIN {X 0,Y 129.866,Z 456.536,A -85,B 0,C 180,E1 -25259.217,E2 -25259.217} C_VEL
LIN {X 0,Y 127.36,Z 458.667,A -85,B 0,C 180,E1 -25261.39,E2 -25261.39} C_VEL
LIN {X 0,Y 123.896,Z 462.647,A -85,B 0,C 180,E1 -25266.604,E2 -25266.604} C_VEL
LIN {X 0,Y 120.936,Z 466.192,A -85,B 0,C 180,E1 -25273.108,E2 -25273.108} C_VEL
LIN {X 0,Y 119.48,Z 468.535,A -85,B 0,C 180,E1 -25279.836,E2 -25279.836} C_VEL
LIN {X 0,Y 119.181,Z 469.721,A -85,B 0,C 180,E1 -25286.619,E2 -25286.619} C_VEL
LIN {X 0,Y 119.332,Z 469.881,A -85,B 0,C 180,E1 -25290,E2 -25290} C_VEL
LIN {X 0,Y 119.204,Z 469.252,A -85,B 0,C 180,E1 -25296.772,E2 -25296.772} C_VEL
LIN {X 0,Y 120.035,Z 467.465,A -85,B 0,C 180,E1 -25303.544,E2 -25303.544} C_VEL
LIN {X 0,Y 122.233,Z 464.508,A -85,B 0,C 180,E1 -25310.181,E2 -25310.181} C_VEL
LIN {X 0,Y 125.799,Z 460.246,A -85,B 0,C 180,E1 -25316.637,E2 -25316.637} C_VEL
LIN {X 0,Y 130.726,Z 454.767,A -85,B 0,C 180,E1 -25322.521,E2 -25322.521} C_VEL
LIN {X 0,Y 137.043,Z 447.732,A -85,B 0,C 180,E1 -25327.981,E2 -25327.981} C_VEL
LIN {X 0,Y 143.323,Z 440.221,A -85,B 0,C 180,E1 -25332.387,E2 -25332.387} C_VEL
LIN {X 0,Y 150.427,Z 431.151,A -85,B 0,C 180,E1 -25336.399,E2 -25336.399} C_VEL
LIN {X 0,Y 158.293,Z 420.269,A -85,B 0,C 180,E1 -25339.985,E2 -25339.985} C_VEL
LIN {X 0,Y 165.519,Z 409.073,A -85,B 0,C 180,E1 -25342.763,E2 -25342.763} C_VEL
LIN {X 0,Y 172.361,Z 396.962,A -85,B 0,C 180,E1 -25345.075,E2 -25345.075} C_VEL
LIN {X 0,Y 178.282,Z 384.737,A -85,B 0,C 180,E1 -25346.897,E2 -25346.897} C_VEL
LIN {X 0,Y 183.644,Z 371.813,A -85,B 0,C 180,E1 -25348.375,E2 -25348.375} C_VEL
LIN {X 0,Y 188.488,Z 357.788,A -85,B 0,C 180,E1 -25349.57,E2 -25349.57} C_VEL
LIN {X 0,Y 192.51,Z 342.756,A -85,B 0,C 180,E1 -25350.514,E2 -25350.514} C_VEL
LIN {X 0,Y 195.42,Z 327.172,A -85,B 0,C 180,E1 -25351.215,E2 -25351.215} C_VEL
LIN {X 0,Y 197.515,Z 308.614,A -85,B 0,C 180,E1 -25351.733,E2 -25351.733} C_VEL
LIN {X 0,Y 201.038,Z 269.751,A -85,B 0,C 180,E1 -25352.75,E2 -25352.75} C_VEL
LIN {X 0,Y 197.388,Z 259.637,A -85,B 0,C 180,E1 -25355.719,E2 -25355.719} C_VEL
LIN {X 0,Y 194.502,Z 252.584,A -85,B 0,C 180,E1 -25358.332,E2 -25358.332} C_VEL
LIN {X 0,Y 191.277,Z 246.856,A -85,B 0,C 180,E1 -25361.524,E2 -25361.524} C_VEL
LIN {X 0,Y 189.607,Z 243.973,A -85,B 0,C 180,E1 -25363.445,E2 -25363.445} C_VEL
LIN {X 0,Y 187.585,Z 240.573,A -85,B 0,C 180,E1 -25366.148,E2 -25366.148} C_VEL
LIN {X 0,Y 185.422,Z 236.75,A -85,B 0,C 180,E1 -25369.904,E2 -25369.904} C_VEL
LIN {X 0,Y 183.604,Z 233.709,A -85,B 0,C 180,E1 -25374.853,E2 -25374.853} C_VEL
LIN {X 0,Y 183.315,Z 232.312,A -85,B 0,C 180,E1 -25376.703,E2 -25376.703} C_VEL
LIN {X 0,Y 183.009,Z 232.005,A -85,B 0,C 180,E1 -25380,E2 -25380} C_VEL
LIN {X 0,Y 183.346,Z 232.475,A -85,B 0,C 180,E1 -25383.984,E2 -25383.984} C_VEL
LIN {X 0,Y 184.698,Z 235.997,A -85,B 0,C 180,E1 -25389.031,E2 -25389.031} C_VEL
LIN {X 0,Y 185.681,Z 237.247,A -85,B 0,C 180,E1 -25391.064,E2 -25391.064} C_VEL
LIN {X 0,Y 188.281,Z 241.767,A -85,B 0,C 180,E1 -25395.285,E2 -25395.285} C_VEL
LIN {X 0,Y 190.679,Z 245.855,A -85,B 0,C 180,E1 -25398.258,E2 -25398.258} C_VEL
LIN {X 0,Y 193.35,Z 250.563,A -85,B 0,C 180,E1 -25401.036,E2 -25401.036} C_VEL
LIN {X 0,Y 196.946,Z 257.262,A -85,B 0,C 180,E1 -25404.229,E2 -25404.229} C_VEL
LIN {X 0,Y 201.189,Z 266.18,A -85,B 0,C 180,E1 -25407.5,E2 -25407.5} C_VEL
LIN {X 0,Y 201.13,Z 268.318,A -85,B 0,C 180,E1 -25407.63,E2 -25407.63} C_VEL
LIN {X 0,Y 196.319,Z 319.085,A -85,B 0,C 180,E1 -25408.982,E2 -25408.982} C_VEL
LIN {X 0,Y 193.568,Z 334.876,A -85,B 0,C 180,E1 -25409.644,E2 -25409.644} C_VEL
LIN {X 0,Y 190.19,Z 348.806,A -85,B 0,C 180,E1 -25410.52,E2 -25410.52} C_VEL
LIN {X 0,Y 185.642,Z 363.38,A -85,B 0,C 180,E1 -25411.798,E2 -25411.798} C_VEL
LIN {X 0,Y 180.291,Z 377.278,A -85,B 0,C 180,E1 -25413.433,E2 -25413.433} C_VEL
LIN {X 0,Y 173.712,Z 391.112,A -85,B 0,C 180,E1 -25415.49,E2 -25415.49} C_VEL
LIN {X 0,Y 166.902,Z 403.312,A -85,B 0,C 180,E1 -25417.858,E2 -25417.858} C_VEL
LIN {X 0,Y 159.813,Z 414.426,A -85,B 0,C 180,E1 -25420.66,E2 -25420.66} C_VEL
LIN {X 0,Y 152.635,Z 424.5,A -85,B 0,C 180,E1 -25423.987,E2 -25423.987} C_VEL
LIN {X 0,Y 147.055,Z 431.724,A -85,B 0,C 180,E1 -25427.076,E2 -25427.076} C_VEL
LIN {X 0,Y 139.547,Z 440.577,A -85,B 0,C 180,E1 -25431.906,E2 -25431.906} C_VEL
LIN {X 0,Y 133.825,Z 446.902,A -85,B 0,C 180,E1 -25436.535,E2 -25436.535} C_VEL
LIN {X 0,Y 128.455,Z 452.704,A -85,B 0,C 180,E1 -25442.287,E2 -25442.287} C_VEL
LIN {X 0,Y 125.227,Z 456.137,A -85,B 0,C 180,E1 -25446.868,E2 -25446.868} C_VEL
LIN {X 0,Y 122.099,Z 459.603,A -85,B 0,C 180,E1 -25453.274,E2 -25453.274} C_VEL
LIN {X 0,Y 120.197,Z 461.887,A -85,B 0,C 180,E1 -25459.897,E2 -25459.897} C_VEL
LIN {X 0,Y 119.437,Z 463.043,A -85,B 0,C 180,E1 -25466.627,E2 -25466.627} C_VEL
LIN {X 0,Y 119.419,Z 463.196,A -85,B 0,C 180,E1 -25470,E2 -25470} C_VEL
LIN {X 0,Y 119.683,Z 462.636,A -85,B 0,C 180,E1 -25476.745,E2 -25476.745} C_VEL
LIN {X 0,Y 120.984,Z 460.963,A -85,B 0,C 180,E1 -25483.436,E2 -25483.436} C_VEL
LIN {X 0,Y 123.403,Z 458.137,A -85,B 0,C 180,E1 -25489.981,E2 -25489.981} C_VEL
LIN {X 0,Y 127.314,Z 454.079,A -85,B 0,C 180,E1 -25496.207,E2 -25496.207} C_VEL
LIN {X 0,Y 132.305,Z 448.698,A -85,B 0,C 180,E1 -25502.087,E2 -25502.087} C_VEL
LIN {X 0,Y 138.604,Z 441.83,A -85,B 0,C 180,E1 -25507.479,E2 -25507.479} C_VEL
